// TIA Portal project "Pepsi_Kem_SindelTCU_2024" (V18)
// Pepsi PID ile calisan akis yonlendirme

(* hardware
DEVICE "S7-1200 station_1"  S7-1200 Station
   slot 0: "Rack_0"  S7-1200 Rack  Rack  V1.0
   slot 1: "PLC_1"  CPU 1215C DC/DC/DC  6ES7 215-1AG40-0XB0  V4.5
   slot 2: "DI 8/DQ 8x24VDC_1"  6ES7 223-1BH32-0XB0  V2.0
   slot 3: "AI 4xTC_1"  SM 1231 AI4 x TC  6ES7 231-5QD32-0XB0  V2.0
DEVICE "GSD device_1"  GSD.Device.PN
   slot 0: "Rack"  Rack  V1.0
   slot 0: "SINAMICS-G120X-PN"  SINAMICS G120X(A) PN V1.0  6SL32xx-xYxxx-xxFx  V1.00
      slot 0: "SINAMICS G120X(A) PN V1.0"  SINAMICS G120X(A) PN V1.0
      slot 1: "PN-IO"  PN-IO
         slot 1: "Port 1"  Port 1
         slot 2: "Port 2"  Port 2
      slot 1: "DRIVE_1"  DRIVE
         slot 0: "Module Access Point"  Module Access Point
         slot 1: "without PROFIsafe"  without PROFIsafe
   slot 2: "Standard telegram 1, PZD-2/2"  Standard telegram 1, PZD-2/2
DEVICE "HMI_1"  KTP400 Basic color PN
   slot 0: "HMI_1"  KTP400 Basic color PN  6AV6 647-0AK11-3AX0  12.0.0.0
   slot 1: "HMI_RT_1"  KTP400 Basic color PN  6AV6 647-0AK11-3AX0  12.0.0.0
   slot 5: "HMI_1.IE_CP_1"  PROFINET Interface  12.0.0.0
      slot 1: "PROFINET Interface_1"  PROFINET Interface
         slot 1: "Port_1"  Port
*)

// ===== PLC "PLC_1"  CPU 1215C DC/DC/DC =====
// protected blocks, not shown: "12_TimeToDint"

VAR_GLOBAL   // PLC tag table "Default tag table"
   "Tag_1" AT %MD200 : Time;
   "Tag_2" AT %M200.0 : Bool;
   "Kalip_Modu" AT %M50.0 : Bool;   // Kalip modu
   "Sirkulasyon Modu" AT %M50.1 : Bool;   // Sirkulasyon modu
   "Seq_KalipVanasi_Kapat" AT %M60.0 : Bool;   // Kalip vanasini kapat
   "Seq_Kalip_Vanasi_Ac" AT %M60.1 : Bool;   // Kalip vanasini ac ve kaliba su gonder
   "System_Byte" AT %MB1 : Byte;
   "FirstScan" AT %M1.0 : Bool;
   "DiagStatusUpdate" AT %M1.1 : Bool;
   "AlwaysTRUE" AT %M1.2 : Bool;
   "AlwaysFALSE" AT %M1.3 : Bool;
   "Clock_Byte" AT %MB0 : Byte;
   "Clock_10Hz" AT %M0.0 : Bool;
   "Clock_5Hz" AT %M0.1 : Bool;
   "Clock_2.5Hz" AT %M0.2 : Bool;
   "Clock_2Hz" AT %M0.3 : Bool;
   "Clock_1.25Hz" AT %M0.4 : Bool;
   "Clock_1Hz" AT %M0.5 : Bool;
   "Clock_0.625Hz" AT %M0.6 : Bool;
   "Clock_0.5Hz" AT %M0.7 : Bool;
   "SuAlmaBaslasin" AT %M2.0 : Bool;   // Su al islemi baslasin
   "Seq_TankVanasi_Ac" AT %M2.1 : Bool;   // 0 - Sirkulasyon | 1- Su al
   "MotorDurdu" AT %M2.2 : Bool;
   "yaslandirmaBaslasin" AT %M2.3 : Bool;
   "Yas_Motor1_kontaktor" AT %M2.4 : Bool;
   "Yas_Motor1_Run" AT %M2.5 : Bool;
   "Yas_Motor2_kontaktor" AT %M3.6 : Bool;
   "Yas_Motor2_Run" AT %M2.6 : Bool;
   "Motor1_kontaktor_Secim1" AT %M2.7 : Bool;
   "Motor1_Run_Secim1" AT %M3.0 : Bool;
   "Motor2_kontaktor_Secim2" AT %M3.1 : Bool;
   "Motor2_Run_Secim2" AT %M3.2 : Bool;
   "PID_Setpoint" AT %MD4 : Real;
   "PID_Mode" AT %MW8 : Int;
   "IsiKontroluBaslasin" AT %M3.3 : Bool;
   "TimeET_demo" AT %MD80 : Time;
   "demoStart" AT %M3.4 : Bool;
   "PID_Tunning_Start" AT %M3.5 : Bool;
   "PID_Manuel_Setpoint" AT %MD10 : Real;
   "BOS" AT %M3.7 : Bool;
   "AlarmSusturSet" AT %M14.0 : Bool;
   "tTermikAtti_AlarmSustur" AT %M14.1 : Bool;
   "Man_Tank_SirDolumVan_Ac" AT %M14.2 : Bool;
   "Man_SirKalip_Van_Kapat" AT %M14.3 : Bool;
   "Man_SirKalip_Van_Ac" AT %M14.4 : Bool;
   "Man_Baypass_Van_Kapat" AT %M14.5 : Bool;
   "Man_Baypass_Van_Ac" AT %M14.6 : Bool;
   "Man_Baypass2_Van_Kapat" AT %M14.7 : Bool;
   "Man_Baypass2_Van_Ac" AT %M15.0 : Bool;
   "Man_Motor1_Run" AT %M15.1 : Bool;
   "Man_Motor2_Run" AT %M15.2 : Bool;
   "Man_Motor1_Kontaktor" AT %M15.3 : Bool;
   "Man_Motor2_Kontaktor" AT %M15.4 : Bool;
   "PID_ModeActive_Auto_Edge" AT %M15.5 : Bool;
   "PID_ModeActive_Man_Edge" AT %M15.6 : Bool;
   "BOS_2" AT %M15.7 : Bool;
   "PID_ModeActive_Edge" AT %M16.0 : Bool;
END_VAR

VAR_GLOBAL   // PLC tag table "Drive"
   "axisOFF1_On" AT %M20.0 : Bool;
   "axisAckError" AT %M20.1 : Bool;
   "axisSpeedSp" AT %MD100 : Real;
   "axisRefSpeed" AT %MD104 : Real;
   "axisHWIDSTW" AT %MW50 : Hw_Io;
   "axisHWIDZSW" AT %MW52 : Hw_Io;
   "axisEnabled" AT %M30.0 : Bool;
   "axisLockout" AT %M30.1 : Bool;
   "axisActVelocity" AT %MD120 : Real;
   "axisError" AT %M30.2 : Bool;
   "axisStatus" AT %MW60 : Word;
   "axisDiagId" AT %MW62 : Word;
END_VAR

VAR_GLOBAL CONSTANT   // PLC tag table "LAcycCom_Common"
   "LACYCCOM_BUFFER_ELEMENTS_UPPER_LIM" : Int := 59;   // Upper limit of request buffer array
END_VAR

VAR_GLOBAL CONSTANT   // PLC tag table "LAcycCom_Drives"
   "LACYCCOM_WRITE_PARAMETERS_UPPER_LIM" : Int := 18;   // Upper limit of write parameters
   "LACYCCOM_READ_PARAMETERS_UPPER_LIM" : Int := 38;   // Upper limit of read parameters
   "LACYCCOM_SILENT_OPERATION_PARAMETERS_UPPER_LIM" : Int := 17;   // Upper limit of parameters in LAcycCom_typeDriveSilentOperation
   "LACYCCOM_NO_COMMAND" : Byte := 16#00;   // No command
   "LACYCCOM_READ_COMMAND" : Byte := 16#01;   // Read command
   "LACYCCOM_WRITE_COMMAND" : Byte := 16#02;   // Write command
   "LACYCCOM_TYPE_ALARM" : SInt := 1;   // Alarm
   "LACYCCOM_TYPE_FAULT" : SInt := 2;   // Fault
   "LACYCCOM_TYPE_SI_MESSAGE" : SInt := 3;   // SI message
   "LACYCCOM_MESSAGES_UPPER_LIM" : Int := 23;   // Upper limit of elements in LAcycCom_typeDriveMessages (fix value)
END_VAR

VAR_GLOBAL   // PLC tag table "IO_INPUT"
   "IN_Acil_stop" AT %I0.0 : Bool;
   "IN_Termik" AT %I0.1 : Bool;
   "IN_Tank_Max" AT %I0.2 : Bool;
   "IN_Tank_Min" AT %I0.3 : Bool;
   "IN_Akis_Valfi" AT %IW64 : Int;   // -- AI 0
   "IN_Giris_Sicakligi" AT %IW96 : Int;   // -- TC 0
   "IN_Cikis_Sicakligi" AT %IW98 : Int;   // -- TC 1
   "IN_Tank_SirkulasyonVeDolumVanasi_Kapali" AT %I0.4 : Bool;
   "IN_Tank_SirkulasyonVeDolumVanasi_Acik" AT %I0.5 : Bool;
   "IN_SirkulasyonVeKalipVanasi_Kapali" AT %I0.6 : Bool;
   "IN_SirkulasyonVeKalipVanasi_Acik" AT %I0.7 : Bool;
   "IN_BaypassVanasi_Kapali" AT %I1.0 : Bool;
   "IN_BaypassVanasi_Acik" AT %I1.1 : Bool;
   "IN_UnknownVana_Kapali" AT %I1.2 : Bool;
   "IN_UnknownVana_Acik" AT %I1.3 : Bool;
   "IN_Remote_Calisiyor" AT %I1.4 : Bool;   // karsi taraftan gelen bilgi
   "IN_Remote_Istek" AT %I1.5 : Bool;   // karsi taraftan gelen kaliba gönder bilgisi
END_VAR

VAR_GLOBAL   // PLC tag table "IO_OUTPUT"
   "OUT_Motor1_Kontaktor" AT %Q0.0 : Bool;   // QK1
   "OUT_Motor2_Kontaktor" AT %Q0.1 : Bool;   // QK2
   "OUT_Tank_SirkulasyonVeDolumVanasi" AT %Q0.2 : Bool;   // V101
   "OUT_SirkulasyonVeKalipVanasi_Kapali" AT %Q0.4 : Bool;   // V201
   "OUT_SirkulasyonVeKalipVanasi_Acik" AT %Q0.5 : Bool;   // V202
   "OUT_BaypassVanasi_Kapali" AT %Q0.6 : Bool;   // V301
   "OUT_BaypassVanasi_Acik" AT %Q0.7 : Bool;   // V302
   "OUT_UnknownVana_Kapali" AT %Q1.0 : Bool;   // V401
   "OUT_UnknownVana_Acik" AT %Q1.1 : Bool;   // V402
   "OUT_Lamba_Yesil" AT %Q2.4 : Bool;
   "OUT_Lamba_Sari" AT %Q2.3 : Bool;
   "OUT_Lamba_Kirmizi" AT %Q2.2 : Bool;
   "OUT_Lamba_Siren" AT %Q2.5 : Bool;
   "OUT_Oransal_Vana" AT %QW64 : Int;
END_VAR

DATA_BLOCK "05_Out_DB"   // DB2
{ S7_Optimized_Access := 'TRUE' }
VERSION : 0.1
// stored: InstanceOfName 05_Out
"05_Out"
BEGIN
END_DATA_BLOCK

DATA_BLOCK "01_Ana Merkez_DB"   // DB3
{ S7_Optimized_Access := 'TRUE' }
VERSION : 0.1
// stored: InstanceOfName 01_Ana Merkez
"01_Ana Merkez"
BEGIN
END_DATA_BLOCK

DATA_BLOCK "04_Manuel_DB"   // DB6
{ S7_Optimized_Access := 'TRUE' }
VERSION : 0.1
// stored: InstanceOfName 04_Manuel
"04_Manuel"
BEGIN
END_DATA_BLOCK

DATA_BLOCK "02_Valf Merkezi_DB"   // DB7
{ S7_Optimized_Access := 'TRUE' }
VERSION : 0.1
// stored: InstanceOfName 02_Valf Merkezi
"02_Valf Merkezi"
BEGIN
END_DATA_BLOCK

DATA_BLOCK "03_Yaslandirma_DB"   // DB8
{ S7_Optimized_Access := 'TRUE' }
VERSION : 0.1
// stored: InstanceOfName 03_Yaslandirma
"03_Yaslandirma"
BEGIN
END_DATA_BLOCK

DATA_BLOCK "07_Alarm_DB"   // DB9
{ S7_Optimized_Access := 'TRUE' }
VERSION : 0.1
// stored: InstanceOfName 07_Alarm
"07_Alarm"
BEGIN
END_DATA_BLOCK

DATA_BLOCK "06_Isı Kontrol Sistemi_DB"   // DB10
{ S7_Optimized_Access := 'TRUE' }
VERSION : 0.1
// stored: InstanceOfName 06_Isı Kontrol Sistemi
"06_Isı Kontrol Sistemi"
BEGIN
END_DATA_BLOCK

// folder: Datablcok

DATA_BLOCK "HMI_Data"   // DB1
{ S7_Optimized_Access := 'TRUE' }
VERSION : 0.1
   VAR
      Buttons : Struct
         Otomatik : Bool;   // otomatik mod
         Manuel : Bool;   // manuel mod
         Start : Bool;   // otomatik mod start
         Stop : Bool;   // otomatik mod stop
         driveAckError : Bool;   // surucu hata reset
         AlarmSustur : Bool;
         ManuelButonlar : Struct
            TankSirDolumVanasi_Ac : Bool;
            SirKalipVanasi_Kapat : Bool;
            SirKalipVanasi_Ac : Bool;
            BaypassVanasi1_Kapat : Bool;
            BaypassVanasi1_Ac : Bool;
            BaypassVanasi2_Kapat : Bool;
            BaypassVanasi2_Ac : Bool;
            Motor1_Run : Bool;
            Motor2_Run : Bool;
         END_STRUCT;
      END_STRUCT;
   END_VAR
   VAR RETAIN
      Datas : Struct
         driveSpeed : Real := 50.0;   // motor istenen hiz
         driveReferenceSp : Real := 100.0;   // motor referans hiz
         istenenYaslandirmaSuresi_saat : Int;   // yaslandirma saat suresi
         istenenYaslandirmaSuresi_dk : Int;   // yaslandirma dakika suresi
         motorTercihi : Byte;   // proses icin motor tercihi
         suAlDelayTime : Time;   // su alma icin bekleme suresi
         IstenenSicaklik : Real;   // Istenen sicaklik
      END_STRUCT;
   END_VAR
   VAR
      Infos : Struct
         AnlikGirisSicakligi : Real;   // Okunan giriş sicaklik
         AnlikCikisSicakligi : Real;   // Okunan cikis sicaklik
         SystemDurumu : String[50] := 'Sistem Basladi';   // Sistem durumu bilgilendirme
         driveError : Bool;   // motor hata var mesajı
         driveEnabled : Bool;   // motor aktif edildi
         driveActVelocity : Real;   // motor anlik hiz
         driveLockout : Bool;   // motor duruyor
         yaslandirmaSuresi_saat : DInt;   // yaslandirma süresi gecen saat suresi
         yaslandirmaSuresi_dk : DInt;   // yaslandirma süresi gecen dakika suresi
         yaslandirmaSuresi_sn : DInt;   // yaslandirma süresi gecen saniye suresi
         yaslandirmaStatus : Struct   // aktif yaslandirma
            sag : Bool;
            sol : Bool;
         END_STRUCT;
         FlowMeterOran : Real;   // Flowmeter akis aciklik orani
         OransalVanaOran : Real;   // Oransal vana aciklik orani
      END_STRUCT;
   END_VAR
BEGIN
END_DATA_BLOCK

DATA_BLOCK "System"   // DB4
{ S7_Optimized_Access := 'TRUE' }
VERSION : 0.1
   VAR
      Auto_Man : Bool;   // 0 - manuel | 1- otomatik
      Step_AnaMerkez : Int;   // Ana calisma modu adim bilgisi
      SysBasladi : Bool;
      YaslandirmaSecimi : Byte;   // Yaslandirma secimi
      Step_Yaslandirma : Byte;   // Yaslandirma islem adimi
      Yaslandirma_Suresi : Time;
      Alarm : Word;   // Alarmlar
   END_VAR
BEGIN
END_DATA_BLOCK

// folder: System blocks/Program resources

DATA_BLOCK "Yas_Motor2_Hold_Timer"   // DB5
{ S7_Optimized_Access := 'TRUE' }
AUTHOR : Simatic
FAMILY : IEC
NAME : IEC_TMR
VERSION : 1.0
// stored: InstanceOfName IEC_TIMER
"IEC_TIMER"
BEGIN
END_DATA_BLOCK

// folder: (top level)

ORGANIZATION_BLOCK "Main"   // OB1, LAD, ProgramCycle
TITLE = "Main Program Sweep (Cycle)"
{ S7_Optimized_Access := 'TRUE' }
VERSION : 0.1
   VAR_INPUT
      Initial_Call : Bool;   // Initial call of this OB
      Remanence : Bool;   // =True, if remanent data are available
   END_VAR
BEGIN

REGION Network 1
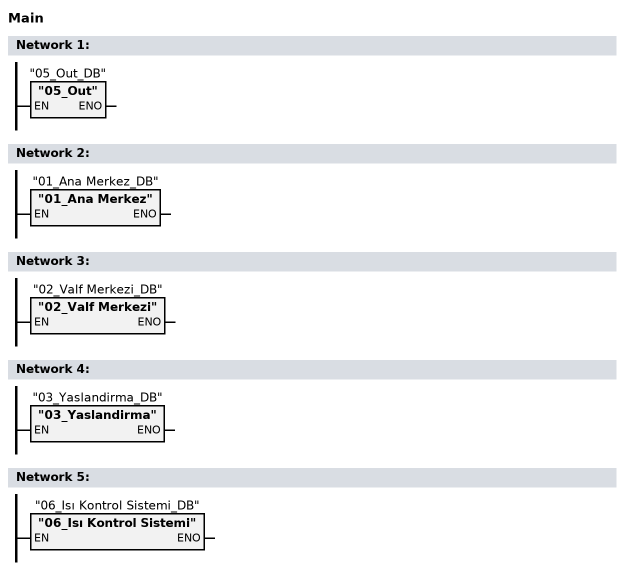
   RUNG wire#powerrail
      "05_Out_DB"()
   END_RUNG
   // the same network as SCL:
   "05_Out_DB"();   // "05_Out"
END_REGION

REGION Network 2
   RUNG wire#powerrail
      "01_Ana Merkez_DB"()
   END_RUNG
   // the same network as SCL:
   "01_Ana Merkez_DB"();   // "01_Ana Merkez"
END_REGION

REGION Network 3
   RUNG wire#powerrail
      "02_Valf Merkezi_DB"()
   END_RUNG
   // the same network as SCL:
   "02_Valf Merkezi_DB"();   // "02_Valf Merkezi"
END_REGION

REGION Network 4
   RUNG wire#powerrail
      "03_Yaslandirma_DB"()
   END_RUNG
   // the same network as SCL:
   "03_Yaslandirma_DB"();   // "03_Yaslandirma"
END_REGION

REGION Network 5
   RUNG wire#powerrail
      "06_Isı Kontrol Sistemi_DB"()
   END_RUNG
   // the same network as SCL:
   "06_Isı Kontrol Sistemi_DB"();   // "06_Isı Kontrol Sistemi"
END_REGION
END_ORGANIZATION_BLOCK

ORGANIZATION_BLOCK "Cyclic interrupt"   // OB30, LAD, CyclicInterrupt
{ S7_Optimized_Access := 'TRUE' }
VERSION : 0.1
   VAR_INPUT
      Initial_Call : Bool;   // Initial call of this OB
      Event_Count : Int;   // Events discarded
   END_VAR
BEGIN

REGION Network 1
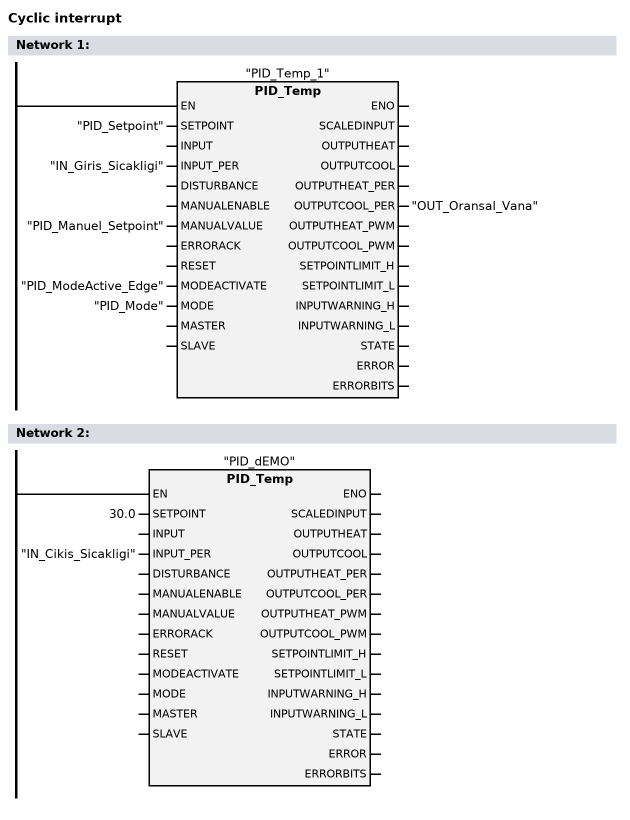
   "PID_Temp_1"(Setpoint := "PID_Setpoint",   // PID_Temp
                Input_PER := "IN_Giris_Sicakligi",
                ManualValue := "PID_Manuel_Setpoint",
                ModeActivate := "PID_ModeActive_Edge",
                Mode := "PID_Mode",
                OutputCool_PER => "OUT_Oransal_Vana");
END_REGION

REGION Network 2
   "PID_dEMO"(Setpoint := 30.0, Input_PER := "IN_Cikis_Sicakligi");   // PID_Temp
END_REGION
END_ORGANIZATION_BLOCK

ORGANIZATION_BLOCK "Diagnostic error interrupt"   // OB82, LAD, DiagnosticErrorInterrupt
{ S7_Optimized_Access := 'TRUE' }
VERSION : 0.1
   VAR_INPUT
      IO_State : Word;   // IO state of the HW object
      LADDR : Hw_Any;   // Hardware identifier
      Channel : UInt;   // Channel number
      MultiError : Bool;   // =true if more than one error is present
   END_VAR
BEGIN
END_ORGANIZATION_BLOCK

ORGANIZATION_BLOCK "Pull or plug of modules"   // OB83, LAD, PullPlug
{ S7_Optimized_Access := 'TRUE' }
VERSION : 0.1
   VAR_INPUT
      LADDR : Hw_Io;   // Hardware identifier
      Event_Class : Byte;   // 16#38/39: module inserted, removed
      Fault_ID : Byte;   // Fault identifier
   END_VAR
BEGIN
END_ORGANIZATION_BLOCK

ORGANIZATION_BLOCK "Rack or station failure"   // OB86, LAD, RackStationFailure
{ S7_Optimized_Access := 'TRUE' }
VERSION : 0.1
   VAR_INPUT
      LADDR : Hw_Device;   // Hardware identifier
      Event_Class : Byte;   // Event class
      Fault_ID : Byte;   // Fault identifier
   END_VAR
BEGIN
END_ORGANIZATION_BLOCK

ORGANIZATION_BLOCK "Task_2"   // OB123, LAD, ProgramCycle
TITLE = "Main Program Sweep (Cycle)"
{ S7_Optimized_Access := 'TRUE' }
VERSION : 0.1
   VAR_INPUT
      Initial_Call : Bool;   // Initial call of this OB
      Remanence : Bool;   // =True, if remanent data are available
   END_VAR
BEGIN

REGION Network 1
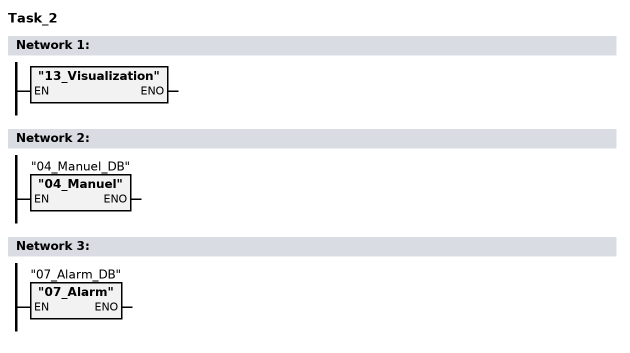
   RUNG wire#powerrail
      "13_Visualization"()
   END_RUNG
   // the same network as SCL:
   "13_Visualization"();
END_REGION

REGION Network 2
   RUNG wire#powerrail
      "04_Manuel_DB"()
   END_RUNG
   // the same network as SCL:
   "04_Manuel_DB"();   // "04_Manuel"
END_REGION

REGION Network 3
   RUNG wire#powerrail
      "07_Alarm_DB"()
   END_RUNG
   // the same network as SCL:
   "07_Alarm_DB"();   // "07_Alarm"
END_REGION
END_ORGANIZATION_BLOCK

// folder: Function

FUNCTION "11_IntToTimer" : Void   // FC1, LAD
{ S7_Optimized_Access := 'TRUE' }
VERSION : 0.1
   VAR_INPUT
      Saat : Int;
      Dakika : Int;
   END_VAR
   VAR_OUTPUT
      HesaplananSure : Time;
   END_VAR
   VAR_TEMP
      tSaat_Dint : DInt;
      tHesaplananSaat : DInt;
      tDakika_Dint : DInt;
      tHesaplananDakika : DInt;
      tHesaplananSure_Dint : DInt;
      tHesaplananSure_Real : Real;
   END_VAR
BEGIN

REGION Network 1
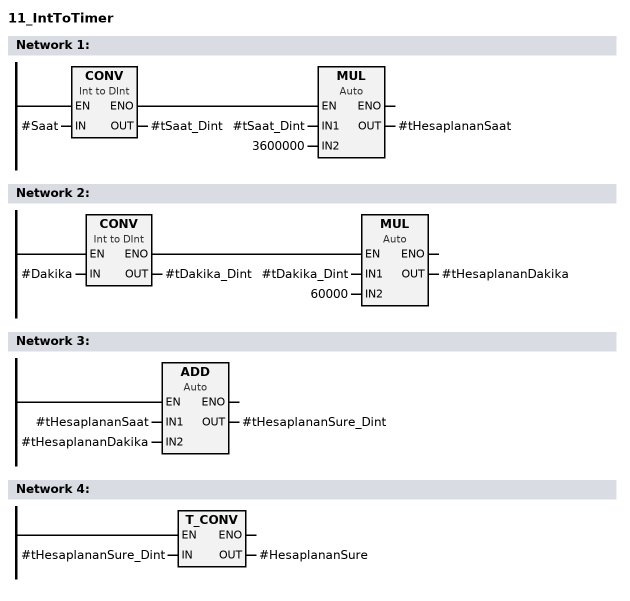
   RUNG wire#powerrail
      { S7_Templates := "[SrcType := Int, DestType := DInt]" } Convert(in := #Saat, out => #tSaat_Dint)
      Mul(in1 := #tSaat_Dint, in2 := 3600000, out => #tHesaplananSaat)
   END_RUNG
   // the same network as SCL:
   #tSaat_Dint := INT_TO_DINT(#Saat);
   #tHesaplananSaat := #tSaat_Dint * 3600000;
END_REGION

REGION Network 2
   RUNG wire#powerrail
      { S7_Templates := "[SrcType := Int, DestType := DInt]" } Convert(in := #Dakika, out => #tDakika_Dint)
      Mul(in1 := #tDakika_Dint, in2 := 60000, out => #tHesaplananDakika)
   END_RUNG
   // the same network as SCL:
   #tDakika_Dint := INT_TO_DINT(#Dakika);
   #tHesaplananDakika := #tDakika_Dint * 60000;
END_REGION

REGION Network 3
   RUNG wire#powerrail
      Add(in1 := #tHesaplananSaat, in2 := #tHesaplananDakika, out => #tHesaplananSure_Dint)
   END_RUNG
   // the same network as SCL:
   #tHesaplananSure_Dint := #tHesaplananSaat + #tHesaplananDakika;
END_REGION

REGION Network 4
   #HesaplananSure := T_CONV(IN := #tHesaplananSure_Dint);
END_REGION
END_FUNCTION

FUNCTION "13_Visualization" : Void   // FC3, LAD
{ S7_Optimized_Access := 'TRUE' }
VERSION : 0.1
// EKRAN BILGILERI VE DONUSUMLERI
   VAR_TEMP
      tGirisSicakligi : Real;
      tCikisSicakligi : Real;
   END_VAR
BEGIN

REGION Network 1 (SCL): Sistem durumu bilgilendirme

   // ana ekran bilgilendirme mesajı
   IF "axisError" THEN
       "HMI_Data".Infos.SystemDurumu := 'Surucu hatasi';
   ELSIF NOT "IN_Termik" THEN
       "HMI_Data".Infos.SystemDurumu := 'Termik hatasi veya 2L+ sigor. kontrol et';
   ELSIF "Kalip_Modu" THEN
       "HMI_Data".Infos.SystemDurumu := 'Kaliba gonderiliyor';
   ELSIF "Sirkulasyon Modu" THEN
       "HMI_Data".Infos.SystemDurumu := 'Sirkulasyon yapiliyor';
   ELSIF NOT "System".Auto_Man THEN
       "HMI_Data".Infos.SystemDurumu := 'Manuel Mod kullanimda';
   END_IF;

   // yaslandirma secimi ekran bilgilendirme
   IF ("System".YaslandirmaSecimi = 0
       AND "System".Step_Yaslandirma = 1)
       OR "System".YaslandirmaSecimi = 1 THEN
       "HMI_Data".Infos.yaslandirmaStatus.sol := true;
       "HMI_Data".Infos.yaslandirmaStatus.sag := FALSE;
   ELSIF ("System".YaslandirmaSecimi = 0
       AND "System".Step_Yaslandirma = 2)
       OR "System".YaslandirmaSecimi = 2 THEN
       "HMI_Data".Infos.yaslandirmaStatus.sol := FALSE;
       "HMI_Data".Infos.yaslandirmaStatus.sag := true;
   END_IF;
END_REGION

REGION Network 2: Akis valfi yuzdesel donusum
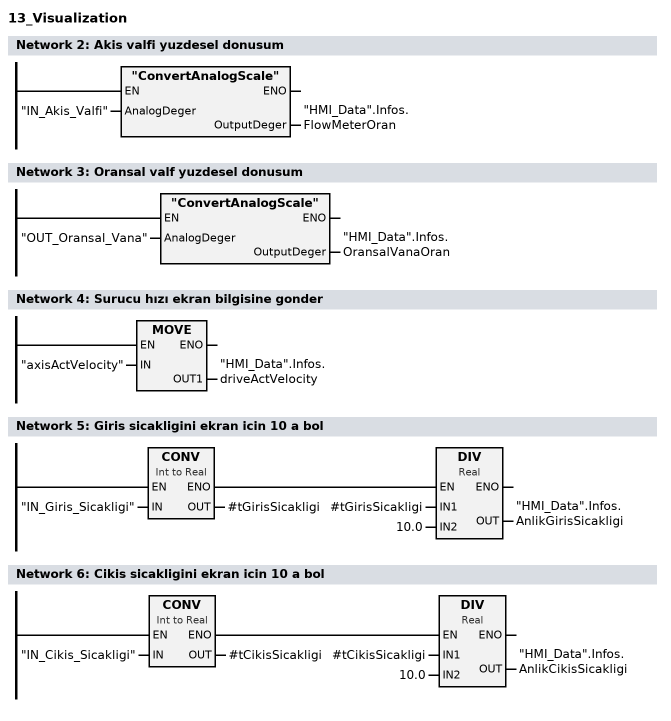
   RUNG wire#powerrail
      "ConvertAnalogScale"(AnalogDeger := "IN_Akis_Valfi", OutputDeger => "HMI_Data".Infos.FlowMeterOran)
   END_RUNG
   // the same network as SCL:
   "ConvertAnalogScale"(AnalogDeger := "IN_Akis_Valfi", OutputDeger => "HMI_Data".Infos.FlowMeterOran);
END_REGION

REGION Network 3: Oransal valf yuzdesel donusum
   RUNG wire#powerrail
      "ConvertAnalogScale"(AnalogDeger := "OUT_Oransal_Vana", OutputDeger => "HMI_Data".Infos.OransalVanaOran)
   END_RUNG
   // the same network as SCL:
   "ConvertAnalogScale"(AnalogDeger := "OUT_Oransal_Vana", OutputDeger => "HMI_Data".Infos.OransalVanaOran);
END_REGION

REGION Network 4: Surucu hızı ekran bilgisine gonder
   RUNG wire#powerrail
      Move(in := "axisActVelocity", out1 => "HMI_Data".Infos.driveActVelocity)
   END_RUNG
   // the same network as SCL:
   "HMI_Data".Infos.driveActVelocity := "axisActVelocity";
END_REGION

REGION Network 5: Giris sicakligini ekran icin 10 a bol
   RUNG wire#powerrail
      { S7_Templates := "[SrcType := Int, DestType := Real]" } Convert(in := "IN_Giris_Sicakligi", out => #tGirisSicakligi)
      { S7_Templates := "SrcType := Real" } Div(in1 := #tGirisSicakligi, in2 := 10.0, out => "HMI_Data".Infos.AnlikGirisSicakligi)
   END_RUNG
   // the same network as SCL:
   #tGirisSicakligi := INT_TO_REAL("IN_Giris_Sicakligi");
   "HMI_Data".Infos.AnlikGirisSicakligi := #tGirisSicakligi / 10.0;
END_REGION

REGION Network 6: Cikis sicakligini ekran icin 10 a bol
   RUNG wire#powerrail
      { S7_Templates := "[SrcType := Int, DestType := Real]" } Convert(in := "IN_Cikis_Sicakligi", out => #tCikisSicakligi)
      { S7_Templates := "SrcType := Real" } Div(in1 := #tCikisSicakligi, in2 := 10.0, out => "HMI_Data".Infos.AnlikCikisSicakligi)
   END_RUNG
   // the same network as SCL:
   #tCikisSicakligi := INT_TO_REAL("IN_Cikis_Sicakligi");
   "HMI_Data".Infos.AnlikCikisSicakligi := #tCikisSicakligi / 10.0;
END_REGION
END_FUNCTION

FUNCTION "ConvertAnalogScale" : Void   // FC4, LAD
{ S7_Optimized_Access := 'TRUE' }
VERSION : 0.1
   VAR_INPUT
      AnalogDeger : Int;
   END_VAR
   VAR_OUTPUT
      OutputDeger : Real;
   END_VAR
   VAR_TEMP
      tRealValue : Real;
      tNorm_Result : Real;
   END_VAR
BEGIN

REGION Network 1
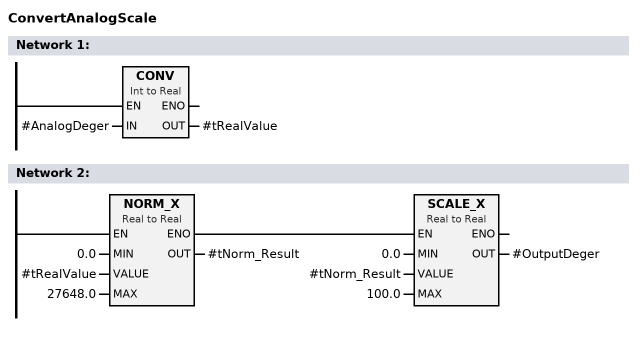
   RUNG wire#powerrail
      { S7_Templates := "[SrcType := Int, DestType := Real]" } Convert(in := #AnalogDeger, out => #tRealValue)
   END_RUNG
   // the same network as SCL:
   #tRealValue := INT_TO_REAL(#AnalogDeger);
END_REGION

REGION Network 2
   RUNG wire#powerrail
      { S7_Templates := "[SrcType := Real, DestType := Real]" } Normalize(min := 0.0, value := #tRealValue, max := 27648.0, out => #tNorm_Result)
      { S7_Templates := "[SrcType := Real, DestType := Real]" } Scale(min := 0.0, value := #tNorm_Result, max := 100.0, out => #OutputDeger)
   END_RUNG
   // the same network as SCL:
   #tNorm_Result := NORM_X(MIN := 0.0, VALUE := #tRealValue, MAX := 27648.0);
   #OutputDeger := SCALE_X(MIN := 0.0, VALUE := #tNorm_Result, MAX := 100.0);
END_REGION
END_FUNCTION

// folder: Function Block

FUNCTION_BLOCK "06_Isı Kontrol Sistemi"   // FB1, LAD
{ S7_Optimized_Access := 'TRUE' }
VERSION : 0.1
// Oransal valfin kontrol edildigi yer
   VAR
      PID_Temp_1 : PID_Temp;
      PID_Compact_1 : PID_Compact;
      ModeActive_M : Bool;
      TP_Timer_Inst : TP_TIME;
      IEC_Timer_0_Instance : TON_TIME;
      IEC_Timer_0_Instance_1 : TP_TIME;
   END_VAR
   VAR_TEMP   // added for the SCL form of the ladder/FBD networks
      _w1 : Bool;
   END_VAR
   // PID_Temp_1.Mode := 4;
BEGIN

REGION Network 1: Oransal valf baslama sarti
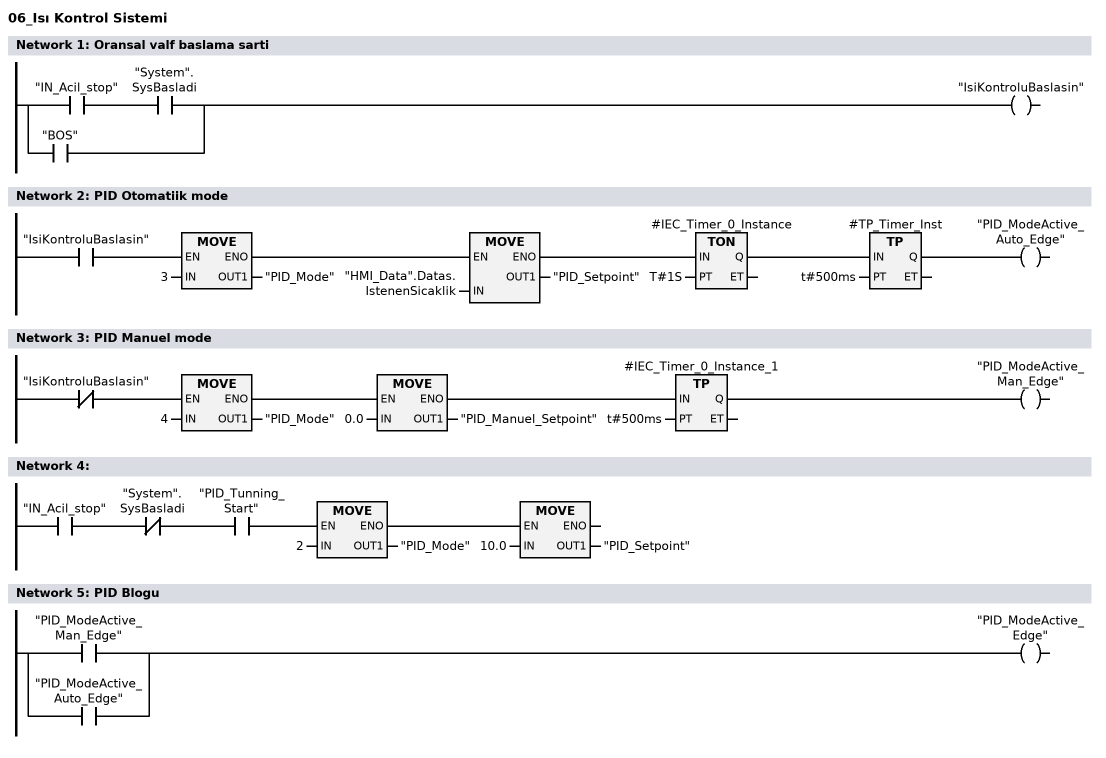
   RUNG wire#powerrail
      Contact( "IN_Acil_stop" )
      Contact( "System".SysBasladi )
      wire#w1
      Coil( "IsiKontroluBaslasin" )
   END_RUNG
   RUNG wire#powerrail
      Contact( "BOS" )
   END_RUNG wire#w1
   // the same network as SCL:
   "IsiKontroluBaslasin" := ("IN_Acil_stop" AND "System".SysBasladi) OR "BOS";
END_REGION

REGION Network 2: PID Otomatiik mode
   IF "IsiKontroluBaslasin" THEN
       "PID_Mode" := 3;
       "PID_Setpoint" := "HMI_Data".Datas.IstenenSicaklik;
   END_IF;
   #IEC_Timer_0_Instance(IN := "IsiKontroluBaslasin", PT := T#1S);   // TON
   #TP_Timer_Inst(IN := #IEC_Timer_0_Instance.Q, PT := t#500ms);   // TP
   "PID_ModeActive_Auto_Edge" := #TP_Timer_Inst.Q;
END_REGION

REGION Network 3: PID Manuel mode
   #_w1 := NOT "IsiKontroluBaslasin";
   IF #_w1 THEN
       "PID_Mode" := 4;
       "PID_Manuel_Setpoint" := 0.0;
   END_IF;
   #IEC_Timer_0_Instance_1(IN := #_w1, PT := t#500ms);   // TP
   "PID_ModeActive_Man_Edge" := #IEC_Timer_0_Instance_1.Q;
END_REGION

REGION Network 4
   RUNG wire#powerrail
      Contact( "IN_Acil_stop" )
      I_Contact( "System".SysBasladi )
      Contact( "PID_Tunning_Start" )
      Move(in := 2, out1 => "PID_Mode")
      Move(in := 10.0, out1 => "PID_Setpoint")
   END_RUNG
   // the same network as SCL:
   IF "IN_Acil_stop" AND NOT "System".SysBasladi AND "PID_Tunning_Start" THEN
       "PID_Mode" := 2;
       "PID_Setpoint" := 10.0;
   END_IF;
END_REGION

REGION Network 5: PID Blogu
   RUNG wire#powerrail
      Contact( "PID_ModeActive_Man_Edge" )
      wire#w1
      Coil( "PID_ModeActive_Edge" )
   END_RUNG
   RUNG wire#powerrail
      Contact( "PID_ModeActive_Auto_Edge" )
   END_RUNG wire#w1
   // the same network as SCL:
   "PID_ModeActive_Edge" := "PID_ModeActive_Man_Edge" OR "PID_ModeActive_Auto_Edge";
END_REGION
END_FUNCTION_BLOCK

FUNCTION_BLOCK "05_Out"   // FB2, LAD
{ S7_Optimized_Access := 'TRUE' }
VERSION : 0.1
   VAR
      SinaSpeed_Instance : SinaSpeed;
   END_VAR
BEGIN

REGION Network 1: Sürücü durdu
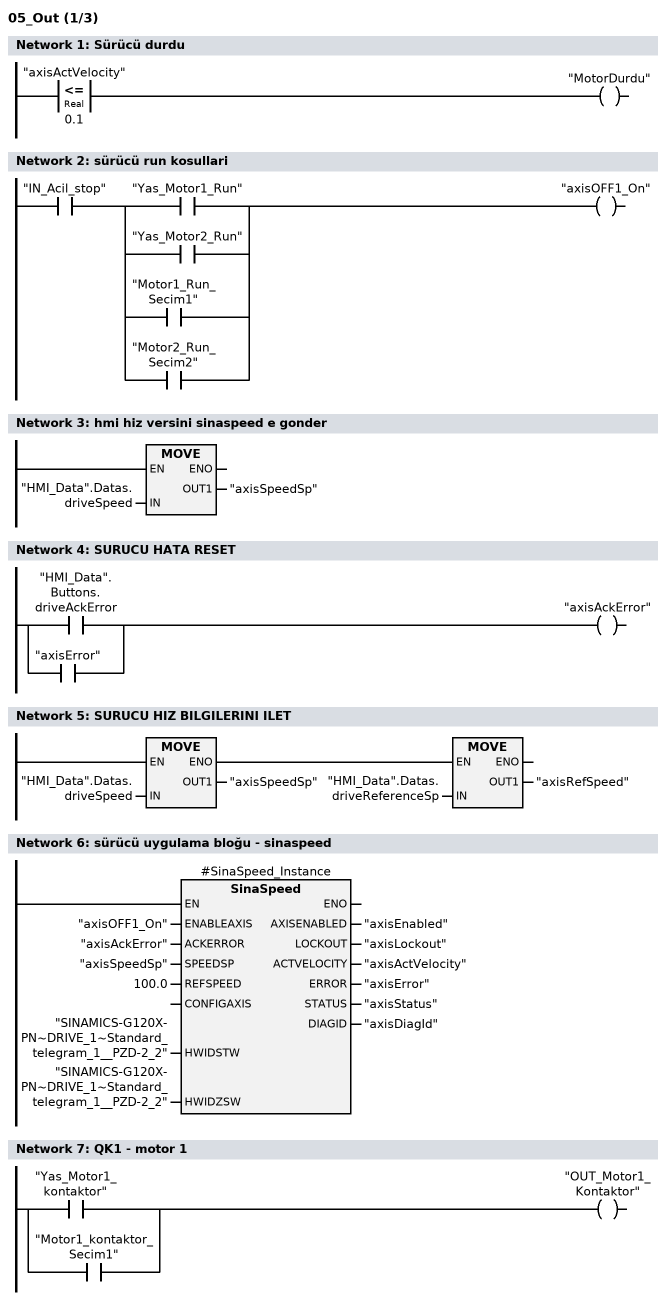
   RUNG wire#powerrail
      { S7_Templates := "SrcType := Real" } LE_Contact(in1 := "axisActVelocity", in2 := 0.1)
      Coil( "MotorDurdu" )
   END_RUNG
   // the same network as SCL:
   "MotorDurdu" := "axisActVelocity" <= 0.1;
END_REGION

REGION Network 2: sürücü run kosullari
   RUNG wire#powerrail
      Contact( "IN_Acil_stop" )
      wire#w1
      Contact( "Yas_Motor1_Run" )
      wire#w2
      Coil( "axisOFF1_On" )
   END_RUNG
   RUNG wire#w1
      Contact( "Yas_Motor2_Run" )
   END_RUNG wire#w2
   RUNG wire#w1
      Contact( "Motor1_Run_Secim1" )
   END_RUNG wire#w2
   RUNG wire#w1
      Contact( "Motor2_Run_Secim2" )
   END_RUNG wire#w2
   // the same network as SCL:
   "axisOFF1_On" := "IN_Acil_stop" AND ("Yas_Motor1_Run" OR "Yas_Motor2_Run" OR "Motor1_Run_Secim1" OR "Motor2_Run_Secim2");
END_REGION

REGION Network 3: hmi hiz versini sinaspeed e gonder
   RUNG wire#powerrail
      Move(in := "HMI_Data".Datas.driveSpeed, out1 => "axisSpeedSp")
   END_RUNG
   // the same network as SCL:
   "axisSpeedSp" := "HMI_Data".Datas.driveSpeed;
END_REGION

REGION Network 4: SURUCU HATA RESET
   RUNG wire#powerrail
      Contact( "HMI_Data".Buttons.driveAckError )
      wire#w1
      Coil( "axisAckError" )
   END_RUNG
   RUNG wire#powerrail
      Contact( "axisError" )
   END_RUNG wire#w1
   // the same network as SCL:
   "axisAckError" := "HMI_Data".Buttons.driveAckError OR "axisError";
END_REGION

REGION Network 5: SURUCU HIZ BILGILERINI ILET
   RUNG wire#powerrail
      Move(in := "HMI_Data".Datas.driveSpeed, out1 => "axisSpeedSp")
      Move(in := "HMI_Data".Datas.driveReferenceSp, out1 => "axisRefSpeed")
   END_RUNG
   // the same network as SCL:
   "axisSpeedSp" := "HMI_Data".Datas.driveSpeed;
   "axisRefSpeed" := "HMI_Data".Datas.driveReferenceSp;
END_REGION

REGION Network 6: sürücü uygulama bloğu - sinaspeed
   #SinaSpeed_Instance(EnableAxis := "axisOFF1_On",   // SinaSpeed
                       AckError := "axisAckError",
                       SpeedSp := "axisSpeedSp",
                       RefSpeed := 100.0,
                       HWIDSTW := "SINAMICS-G120X-PN~DRIVE_1~Standard_telegram_1__PZD-2_2",
                       HWIDZSW := "SINAMICS-G120X-PN~DRIVE_1~Standard_telegram_1__PZD-2_2",
                       AxisEnabled => "axisEnabled",
                       Lockout => "axisLockout",
                       ActVelocity => "axisActVelocity",
                       Error => "axisError",
                       Status => "axisStatus",
                       DiagId => "axisDiagId");
END_REGION

REGION Network 7: QK1 - motor 1
   RUNG wire#powerrail
      Contact( "Yas_Motor1_kontaktor" )
      wire#w1
      Coil( "OUT_Motor1_Kontaktor" )
   END_RUNG
   RUNG wire#powerrail
      Contact( "Motor1_kontaktor_Secim1" )
   END_RUNG wire#w1
   // the same network as SCL:
   "OUT_Motor1_Kontaktor" := "Yas_Motor1_kontaktor" OR "Motor1_kontaktor_Secim1";
END_REGION

REGION Network 8: QK2 - motor 2
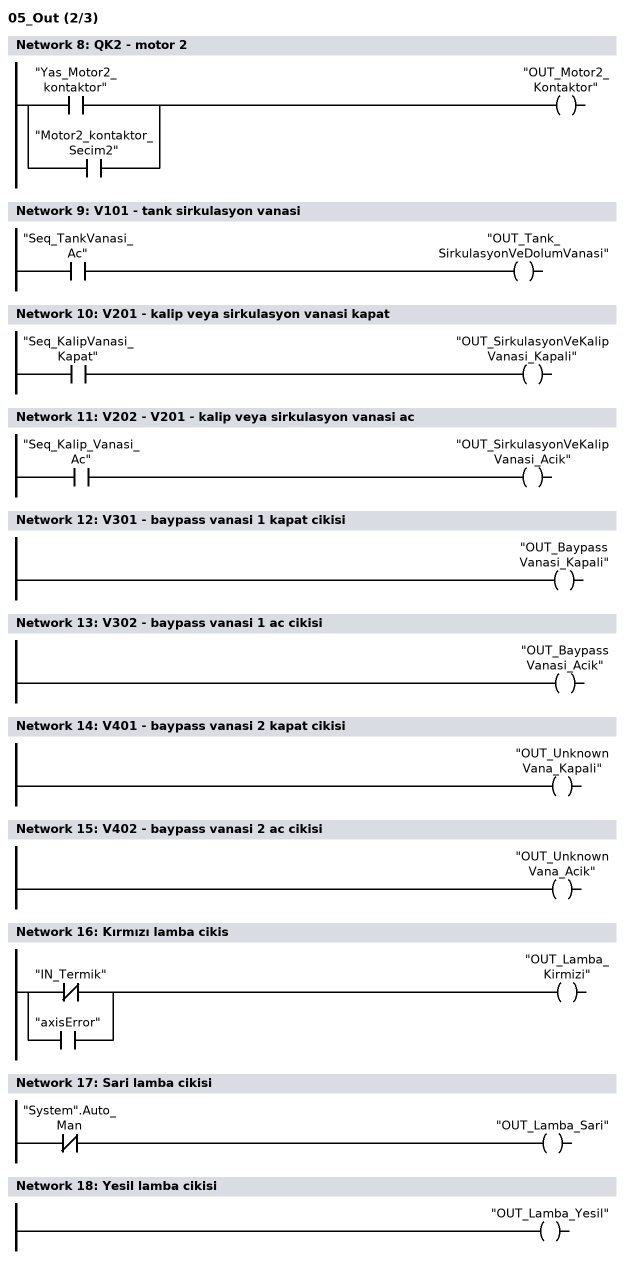
   RUNG wire#powerrail
      Contact( "Yas_Motor2_kontaktor" )
      wire#w1
      Coil( "OUT_Motor2_Kontaktor" )
   END_RUNG
   RUNG wire#powerrail
      Contact( "Motor2_kontaktor_Secim2" )
   END_RUNG wire#w1
   // the same network as SCL:
   "OUT_Motor2_Kontaktor" := "Yas_Motor2_kontaktor" OR "Motor2_kontaktor_Secim2";
END_REGION

REGION Network 9: V101 - tank sirkulasyon vanasi
   RUNG wire#powerrail
      Contact( "Seq_TankVanasi_Ac" )
      Coil( "OUT_Tank_SirkulasyonVeDolumVanasi" )
   END_RUNG
   // the same network as SCL:
   "OUT_Tank_SirkulasyonVeDolumVanasi" := "Seq_TankVanasi_Ac";
END_REGION

REGION Network 10: V201 - kalip veya sirkulasyon vanasi kapat
   RUNG wire#powerrail
      Contact( "Seq_KalipVanasi_Kapat" )
      Coil( "OUT_SirkulasyonVeKalipVanasi_Kapali" )
   END_RUNG
   // the same network as SCL:
   "OUT_SirkulasyonVeKalipVanasi_Kapali" := "Seq_KalipVanasi_Kapat";
END_REGION

REGION Network 11: V202 - V201 - kalip veya sirkulasyon vanasi ac
   RUNG wire#powerrail
      Contact( "Seq_Kalip_Vanasi_Ac" )
      Coil( "OUT_SirkulasyonVeKalipVanasi_Acik" )
   END_RUNG
   // the same network as SCL:
   "OUT_SirkulasyonVeKalipVanasi_Acik" := "Seq_Kalip_Vanasi_Ac";
END_REGION

REGION Network 12: V301 - baypass vanasi 1 kapat cikisi
   RUNG wire#powerrail
      Coil( "OUT_BaypassVanasi_Kapali" )
   END_RUNG
   // the same network as SCL:
   "OUT_BaypassVanasi_Kapali" := TRUE;
END_REGION

REGION Network 13: V302 - baypass vanasi 1 ac cikisi
   RUNG wire#powerrail
      Coil( "OUT_BaypassVanasi_Acik" )
   END_RUNG
   // the same network as SCL:
   "OUT_BaypassVanasi_Acik" := TRUE;
END_REGION

REGION Network 14: V401 - baypass vanasi 2 kapat cikisi
   RUNG wire#powerrail
      Coil( "OUT_UnknownVana_Kapali" )
   END_RUNG
   // the same network as SCL:
   "OUT_UnknownVana_Kapali" := TRUE;
END_REGION

REGION Network 15: V402 - baypass vanasi 2 ac cikisi
   RUNG wire#powerrail
      Coil( "OUT_UnknownVana_Acik" )
   END_RUNG
   // the same network as SCL:
   "OUT_UnknownVana_Acik" := TRUE;
END_REGION

REGION Network 16: Kırmızı lamba cikis
   RUNG wire#powerrail
      I_Contact( "IN_Termik" )
      wire#w1
      Coil( "OUT_Lamba_Kirmizi" )
   END_RUNG
   RUNG wire#powerrail
      Contact( "axisError" )
   END_RUNG wire#w1
   // the same network as SCL:
   "OUT_Lamba_Kirmizi" := NOT "IN_Termik" OR "axisError";
END_REGION

REGION Network 17: Sari lamba cikisi
   RUNG wire#powerrail
      I_Contact( "System".Auto_Man )
      Coil( "OUT_Lamba_Sari" )
   END_RUNG
   // the same network as SCL:
   "OUT_Lamba_Sari" := NOT "System".Auto_Man;
END_REGION

REGION Network 18: Yesil lamba cikisi
   RUNG wire#powerrail
      Coil( "OUT_Lamba_Yesil" )
   END_RUNG
   // the same network as SCL:
   "OUT_Lamba_Yesil" := TRUE;
END_REGION

REGION Network 19: Siren lamba cikisi
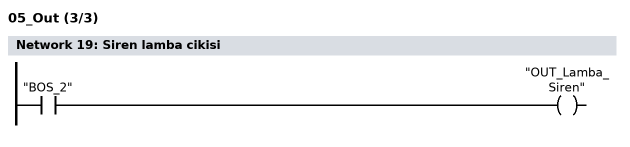
   RUNG wire#powerrail
      Contact( "BOS_2" )
      Coil( "OUT_Lamba_Siren" )
   END_RUNG
   // the same network as SCL:
   "OUT_Lamba_Siren" := "BOS_2";
END_REGION
END_FUNCTION_BLOCK

FUNCTION_BLOCK "07_Alarm"   // FB3, LAD
{ S7_Optimized_Access := 'TRUE' }
VERSION : 0.1
   VAR
      TankDolumVanasi_Inst : TON_TIME;
      KalipDolumVanasi_Inst : TON_TIME;
      BypassVanasi_Inst : TON_TIME;
      BypassVanasi2_Inst : TON_TIME;
      ResetTrig : Bool;
      ResetTrig2 : Bool;
      Manuel_M : Bool;
      Oto_M : Bool;
      Start_M : Bool;
      Stop_M : Bool;
   END_VAR
   VAR_TEMP   // added for the SCL form of the ladder/FBD networks
      _w1 : Bool;
      _w2 : Bool;
      _w3 : Bool;
      _w4 : Bool;
   END_VAR
BEGIN

REGION Network 1: Surucu hata
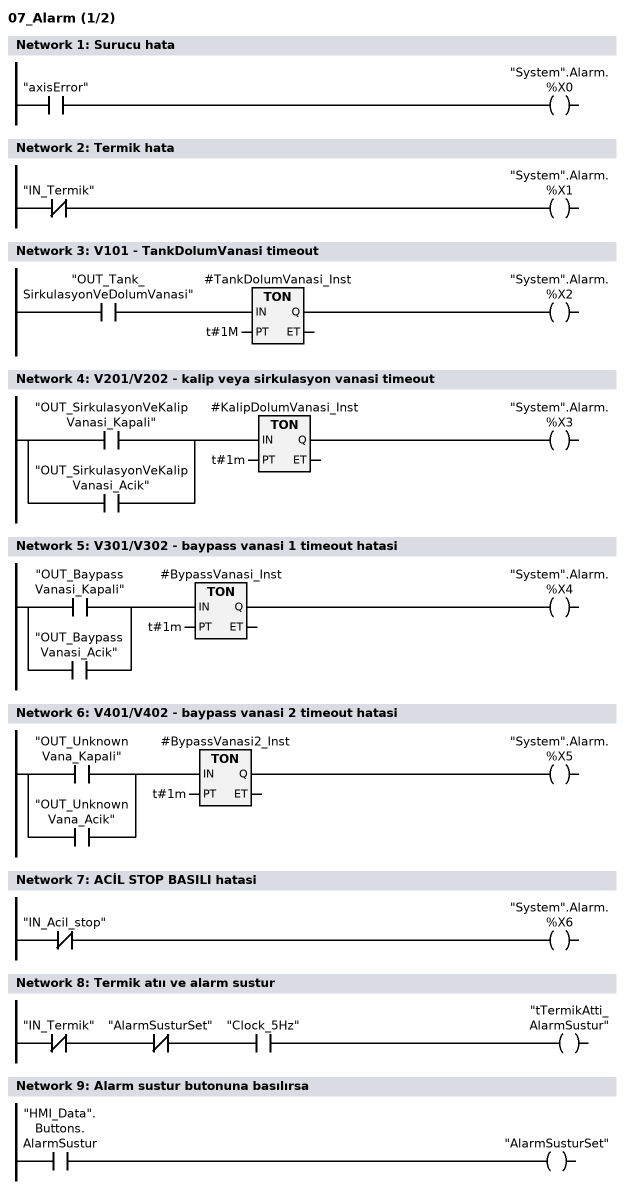
   RUNG wire#powerrail
      Contact( "axisError" )
      Coil( "System".Alarm.%X0 )
   END_RUNG
   // the same network as SCL:
   "System".Alarm.%X0 := "axisError";
END_REGION

REGION Network 2: Termik hata
   RUNG wire#powerrail
      I_Contact( "IN_Termik" )
      Coil( "System".Alarm.%X1 )
   END_RUNG
   // the same network as SCL:
   "System".Alarm.%X1 := NOT "IN_Termik";
END_REGION

REGION Network 3: V101 - TankDolumVanasi timeout
   #TankDolumVanasi_Inst(IN := "OUT_Tank_SirkulasyonVeDolumVanasi", PT := t#1M);   // TON
   "System".Alarm.%X2 := #TankDolumVanasi_Inst.Q;
END_REGION

REGION Network 4: V201/V202 - kalip veya sirkulasyon vanasi timeout
   #KalipDolumVanasi_Inst(IN := "OUT_SirkulasyonVeKalipVanasi_Kapali" OR "OUT_SirkulasyonVeKalipVanasi_Acik",   // TON
                          PT := t#1m);
   "System".Alarm.%X3 := #KalipDolumVanasi_Inst.Q;
END_REGION

REGION Network 5: V301/V302 - baypass vanasi 1 timeout hatasi
   #BypassVanasi_Inst(IN := "OUT_BaypassVanasi_Kapali" OR "OUT_BaypassVanasi_Acik", PT := t#1m);   // TON
   "System".Alarm.%X4 := #BypassVanasi_Inst.Q;
END_REGION

REGION Network 6: V401/V402 - baypass vanasi 2 timeout hatasi
   #BypassVanasi2_Inst(IN := "OUT_UnknownVana_Kapali" OR "OUT_UnknownVana_Acik", PT := t#1m);   // TON
   "System".Alarm.%X5 := #BypassVanasi2_Inst.Q;
END_REGION

REGION Network 7: ACİL STOP BASILI hatasi
   RUNG wire#powerrail
      I_Contact( "IN_Acil_stop" )
      Coil( "System".Alarm.%X6 )
   END_RUNG
   // the same network as SCL:
   "System".Alarm.%X6 := NOT "IN_Acil_stop";
END_REGION

REGION Network 8: Termik atıı ve alarm sustur
   RUNG wire#powerrail
      I_Contact( "IN_Termik" )
      I_Contact( "AlarmSusturSet" )
      Contact( "Clock_5Hz" )
      Coil( "tTermikAtti_AlarmSustur" )
   END_RUNG
   // the same network as SCL:
   "tTermikAtti_AlarmSustur" := NOT "IN_Termik" AND NOT "AlarmSusturSet" AND "Clock_5Hz";
END_REGION

REGION Network 9: Alarm sustur butonuna basılırsa
   RUNG wire#powerrail
      Contact( "HMI_Data".Buttons.AlarmSustur )
      Coil( "AlarmSusturSet" )
   END_RUNG
   // the same network as SCL:
   "AlarmSusturSet" := "HMI_Data".Buttons.AlarmSustur;
END_REGION

REGION Network 10: Alarm sustur bitini resetle
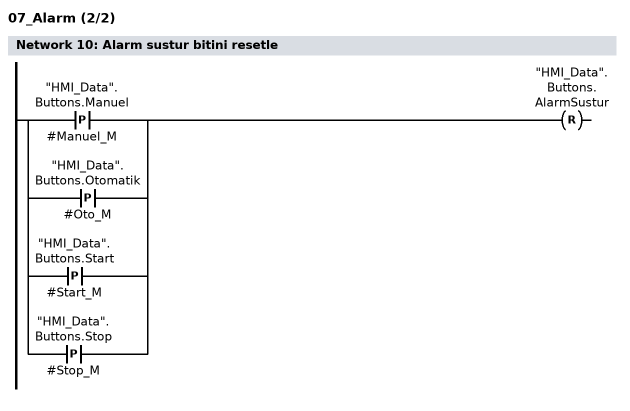
   RUNG wire#powerrail
      P_Contact(operand := "HMI_Data".Buttons.Manuel, bit := #Manuel_M)
      wire#w1
      R_Coil( "HMI_Data".Buttons.AlarmSustur )
   END_RUNG
   RUNG wire#powerrail
      P_Contact(operand := "HMI_Data".Buttons.Otomatik, bit := #Oto_M)
   END_RUNG wire#w1
   RUNG wire#powerrail
      P_Contact(operand := "HMI_Data".Buttons.Start, bit := #Start_M)
   END_RUNG wire#w1
   RUNG wire#powerrail
      P_Contact(operand := "HMI_Data".Buttons.Stop, bit := #Stop_M)
   END_RUNG wire#w1
   // the same network as SCL:
   #_w1 := "HMI_Data".Buttons.Manuel AND NOT #Manuel_M;   // rising edge of "HMI_Data".Buttons.Manuel
   #Manuel_M := "HMI_Data".Buttons.Manuel;
   #_w2 := "HMI_Data".Buttons.Otomatik AND NOT #Oto_M;   // rising edge of "HMI_Data".Buttons.Otomatik
   #Oto_M := "HMI_Data".Buttons.Otomatik;
   #_w3 := "HMI_Data".Buttons.Start AND NOT #Start_M;   // rising edge of "HMI_Data".Buttons.Start
   #Start_M := "HMI_Data".Buttons.Start;
   #_w4 := "HMI_Data".Buttons.Stop AND NOT #Stop_M;   // rising edge of "HMI_Data".Buttons.Stop
   #Stop_M := "HMI_Data".Buttons.Stop;
   IF #_w1 OR #_w2 OR #_w3 OR #_w4 THEN "HMI_Data".Buttons.AlarmSustur := FALSE; END_IF;
END_REGION
END_FUNCTION_BLOCK

FUNCTION_BLOCK "01_Ana Merkez"   // FB4, LAD
{ S7_Optimized_Access := 'TRUE' }
VERSION : 0.1
BEGIN

REGION Network 1
   // otomatik baslama icin gerekli kontroller
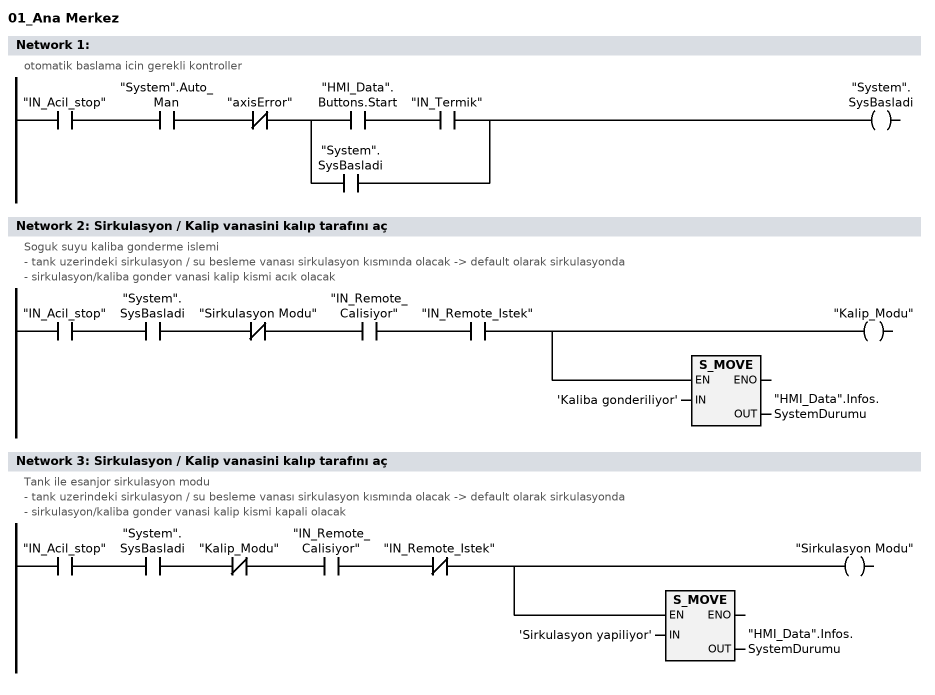
   RUNG wire#powerrail
      Contact( "IN_Acil_stop" )
      Contact( "System".Auto_Man )
      I_Contact( "axisError" )
      wire#w1
      Contact( "HMI_Data".Buttons.Start )
      Contact( "IN_Termik" )
      wire#w2
      Coil( "System".SysBasladi )
   END_RUNG
   RUNG wire#w1
      Contact( "System".SysBasladi )
   END_RUNG wire#w2
   // the same network as SCL:
   "System".SysBasladi := "IN_Acil_stop" AND "System".Auto_Man AND NOT "axisError" AND (("HMI_Data".Buttons.Start AND "IN_Termik") OR "System".SysBasladi);
END_REGION

REGION Network 2: Sirkulasyon / Kalip vanasini kalıp tarafını aç
   // Soguk suyu kaliba gonderme islemi
   // - tank uzerindeki sirkulasyon / su besleme vanası sirkulasyon kısmında olacak -> default olarak sirkulasyonda
   // - sirkulasyon/kaliba gonder vanasi kalip kismi acık olacak
   RUNG wire#powerrail
      Contact( "IN_Acil_stop" )
      Contact( "System".SysBasladi )
      I_Contact( "Sirkulasyon Modu" )
      Contact( "IN_Remote_Calisiyor" )
      Contact( "IN_Remote_Istek" )
      wire#w1
      Coil( "Kalip_Modu" )
   END_RUNG
   RUNG wire#w1
      S_Move(in := 'Kaliba gonderiliyor', out => "HMI_Data".Infos.SystemDurumu)
   END_RUNG
   // the same network as SCL:
   "Kalip_Modu" := "IN_Acil_stop" AND "System".SysBasladi AND NOT "Sirkulasyon Modu" AND "IN_Remote_Calisiyor" AND "IN_Remote_Istek";
   IF "Kalip_Modu" THEN "HMI_Data".Infos.SystemDurumu := 'Kaliba gonderiliyor'; END_IF;
END_REGION

REGION Network 3: Sirkulasyon / Kalip vanasini kalıp tarafını aç
   // Tank ile esanjor sirkulasyon modu
   // - tank uzerindeki sirkulasyon / su besleme vanası sirkulasyon kısmında olacak -> default olarak sirkulasyonda
   // - sirkulasyon/kaliba gonder vanasi kalip kismi kapali olacak
   RUNG wire#powerrail
      Contact( "IN_Acil_stop" )
      Contact( "System".SysBasladi )
      I_Contact( "Kalip_Modu" )
      Contact( "IN_Remote_Calisiyor" )
      I_Contact( "IN_Remote_Istek" )
      wire#w1
      Coil( "Sirkulasyon Modu" )
   END_RUNG
   RUNG wire#w1
      S_Move(in := 'Sirkulasyon yapiliyor', out => "HMI_Data".Infos.SystemDurumu)
   END_RUNG
   // the same network as SCL:
   "Sirkulasyon Modu" := "IN_Acil_stop" AND "System".SysBasladi AND NOT "Kalip_Modu" AND "IN_Remote_Calisiyor" AND NOT "IN_Remote_Istek";
   IF "Sirkulasyon Modu" THEN "HMI_Data".Infos.SystemDurumu := 'Sirkulasyon yapiliyor'; END_IF;
END_REGION
END_FUNCTION_BLOCK

FUNCTION_BLOCK "02_Valf Merkezi"   // FB5, LAD
{ S7_Optimized_Access := 'TRUE' }
VERSION : 0.1
// Sirkulasyon Modu vana kontrolleri
// 
// --------------BYPASS VANALARI EKLENECEK---------------------------
   VAR
      SuAlTimer_Inst : TON_TIME;
      SuAlTimer2_Inst : TON_TIME;
   END_VAR
   VAR_TEMP   // added for the SCL form of the ladder/FBD networks
      _w1 : Bool;
   END_VAR
BEGIN

REGION Network 1: Sirkulasyon Modu -> kalip vanasini kapat
   // Kalip vanasi kapali -> sirkulasyon yapar
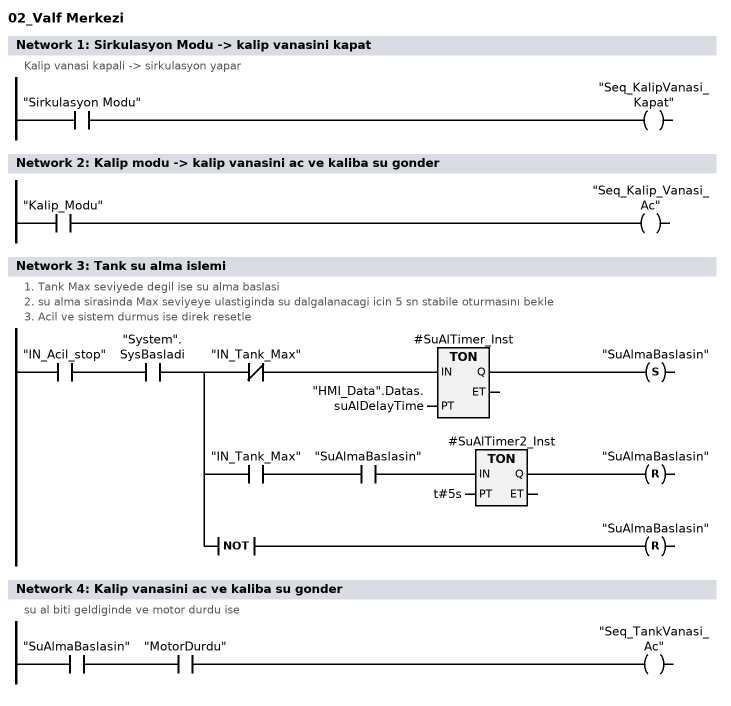
   RUNG wire#powerrail
      Contact( "Sirkulasyon Modu" )
      Coil( "Seq_KalipVanasi_Kapat" )
   END_RUNG
   // the same network as SCL:
   "Seq_KalipVanasi_Kapat" := "Sirkulasyon Modu";
END_REGION

REGION Network 2: Kalip modu -> kalip vanasini ac ve kaliba su gonder
   RUNG wire#powerrail
      Contact( "Kalip_Modu" )
      Coil( "Seq_Kalip_Vanasi_Ac" )
   END_RUNG
   // the same network as SCL:
   "Seq_Kalip_Vanasi_Ac" := "Kalip_Modu";
END_REGION

REGION Network 3: Tank su alma islemi
   // 1. Tank Max seviyede degil ise su alma baslasi
   // 2. su alma sirasinda Max seviyeye ulastiginda su dalgalanacagi icin 5 sn stabile oturmasını bekle
   // 3. Acil ve sistem durmus ise direk resetle
   #_w1 := "IN_Acil_stop" AND "System".SysBasladi;
   #SuAlTimer_Inst(IN := #_w1 AND NOT "IN_Tank_Max", PT := "HMI_Data".Datas.suAlDelayTime);   // TON
   IF #SuAlTimer_Inst.Q THEN "SuAlmaBaslasin" := TRUE; END_IF;
   #SuAlTimer2_Inst(IN := #_w1 AND "IN_Tank_Max" AND "SuAlmaBaslasin", PT := t#5s);   // TON
   IF #SuAlTimer2_Inst.Q THEN "SuAlmaBaslasin" := FALSE; END_IF;
   IF NOT #_w1 THEN "SuAlmaBaslasin" := FALSE; END_IF;
END_REGION

REGION Network 4: Kalip vanasini ac ve kaliba su gonder
   // su al biti geldiginde ve motor durdu ise
   RUNG wire#powerrail
      Contact( "SuAlmaBaslasin" )
      Contact( "MotorDurdu" )
      Coil( "Seq_TankVanasi_Ac" )
   END_RUNG
   // the same network as SCL:
   "Seq_TankVanasi_Ac" := "SuAlmaBaslasin" AND "MotorDurdu";
END_REGION
END_FUNCTION_BLOCK

FUNCTION_BLOCK "03_Yaslandirma"   // FB6, LAD
{ S7_Optimized_Access := 'TRUE' }
VERSION : 0.1
   VAR
      Yas_Motor1_Timer : TON_TIME;
      Yas_Moto1_Hold_Timer : TON_TIME;
      Motor1_Run_Delay : TON_TIME;
      Motor2_Run_Delay : TON_TIME;
      Yas_Motor2_Timer : TON_TIME;
      Yas_Secim1_Motor_Timer : TON_TIME;
      Yas_Secim2_Motor_Timer : TON_TIME;
      IEC_Timer_0_Instance : TON_TIME;
      IEC_Timer_0_Instance_1 : TON_TIME;
   END_VAR
   VAR_TEMP
      Yas_Motor1_TimeET : Time;
      Yas_Motor2_TimeET : Time;
   END_VAR
BEGIN

REGION Network 1: eKRAN SAAT ve DAKIKA degerini TIME 'A DONUSTUR
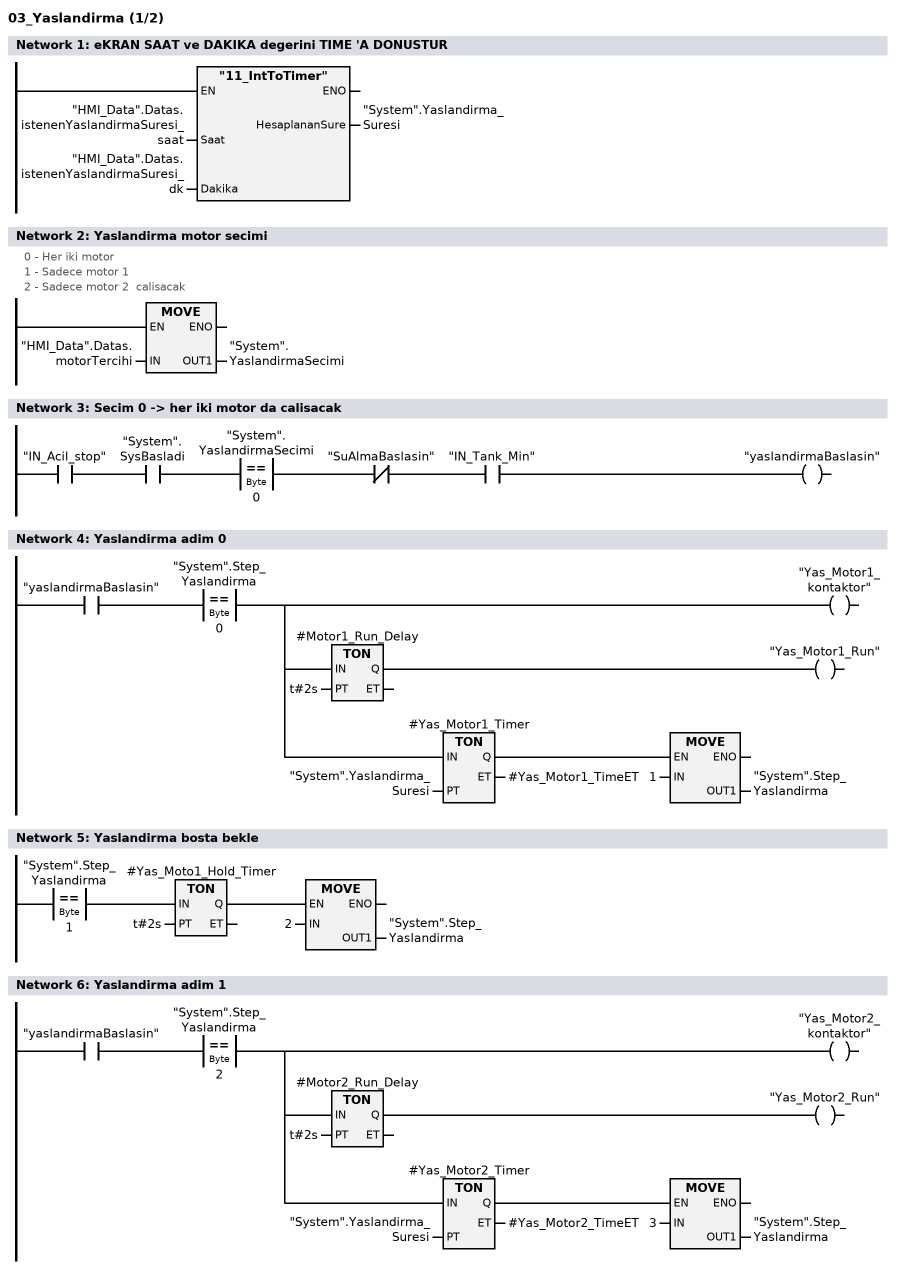
   RUNG wire#powerrail
      "11_IntToTimer"(Saat := "HMI_Data".Datas.istenenYaslandirmaSuresi_saat, Dakika := "HMI_Data".Datas.istenenYaslandirmaSuresi_dk, HesaplananSure => "System".Yaslandirma_Suresi)
   END_RUNG
   // the same network as SCL:
   "11_IntToTimer"(Saat := "HMI_Data".Datas.istenenYaslandirmaSuresi_saat,
                   Dakika := "HMI_Data".Datas.istenenYaslandirmaSuresi_dk,
                   HesaplananSure => "System".Yaslandirma_Suresi);
END_REGION

REGION Network 2: Yaslandirma motor secimi
   // 0 - Her iki motor
   // 1 - Sadece motor 1 
   // 2 - Sadece motor 2  calisacak
   RUNG wire#powerrail
      Move(in := "HMI_Data".Datas.motorTercihi, out1 => "System".YaslandirmaSecimi)
   END_RUNG
   // the same network as SCL:
   "System".YaslandirmaSecimi := "HMI_Data".Datas.motorTercihi;
END_REGION

REGION Network 3: Secim 0 -> her iki motor da calisacak
   RUNG wire#powerrail
      Contact( "IN_Acil_stop" )
      Contact( "System".SysBasladi )
      { S7_Templates := "SrcType := Byte" } EQ_Contact(in1 := "System".YaslandirmaSecimi, in2 := 0)
      I_Contact( "SuAlmaBaslasin" )
      Contact( "IN_Tank_Min" )
      Coil( "yaslandirmaBaslasin" )
   END_RUNG
   // the same network as SCL:
   "yaslandirmaBaslasin" := "IN_Acil_stop" AND "System".SysBasladi AND ("System".YaslandirmaSecimi = 0) AND NOT "SuAlmaBaslasin" AND "IN_Tank_Min";
END_REGION

REGION Network 4: Yaslandirma adim 0
   "Yas_Motor1_kontaktor" := "yaslandirmaBaslasin" AND ("System".Step_Yaslandirma = 0);
   #Motor1_Run_Delay(IN := "Yas_Motor1_kontaktor", PT := t#2s);   // TON
   "Yas_Motor1_Run" := #Motor1_Run_Delay.Q;
   #Yas_Motor1_Timer(IN := "Yas_Motor1_kontaktor", PT := "System".Yaslandirma_Suresi, ET => #Yas_Motor1_TimeET);   // TON
   IF #Yas_Motor1_Timer.Q THEN "System".Step_Yaslandirma := 1; END_IF;
END_REGION

REGION Network 5: Yaslandirma bosta bekle
   #Yas_Moto1_Hold_Timer(IN := "System".Step_Yaslandirma = 1, PT := t#2s);   // TON
   IF #Yas_Moto1_Hold_Timer.Q THEN "System".Step_Yaslandirma := 2; END_IF;
END_REGION

REGION Network 6: Yaslandirma adim 1
   "Yas_Motor2_kontaktor" := "yaslandirmaBaslasin" AND ("System".Step_Yaslandirma = 2);
   #Motor2_Run_Delay(IN := "Yas_Motor2_kontaktor", PT := t#2s);   // TON
   "Yas_Motor2_Run" := #Motor2_Run_Delay.Q;
   #Yas_Motor2_Timer(IN := "Yas_Motor2_kontaktor", PT := "System".Yaslandirma_Suresi, ET => #Yas_Motor2_TimeET);   // TON
   IF #Yas_Motor2_Timer.Q THEN "System".Step_Yaslandirma := 3; END_IF;
END_REGION

REGION Network 7: Yaslandirma bosta bekle
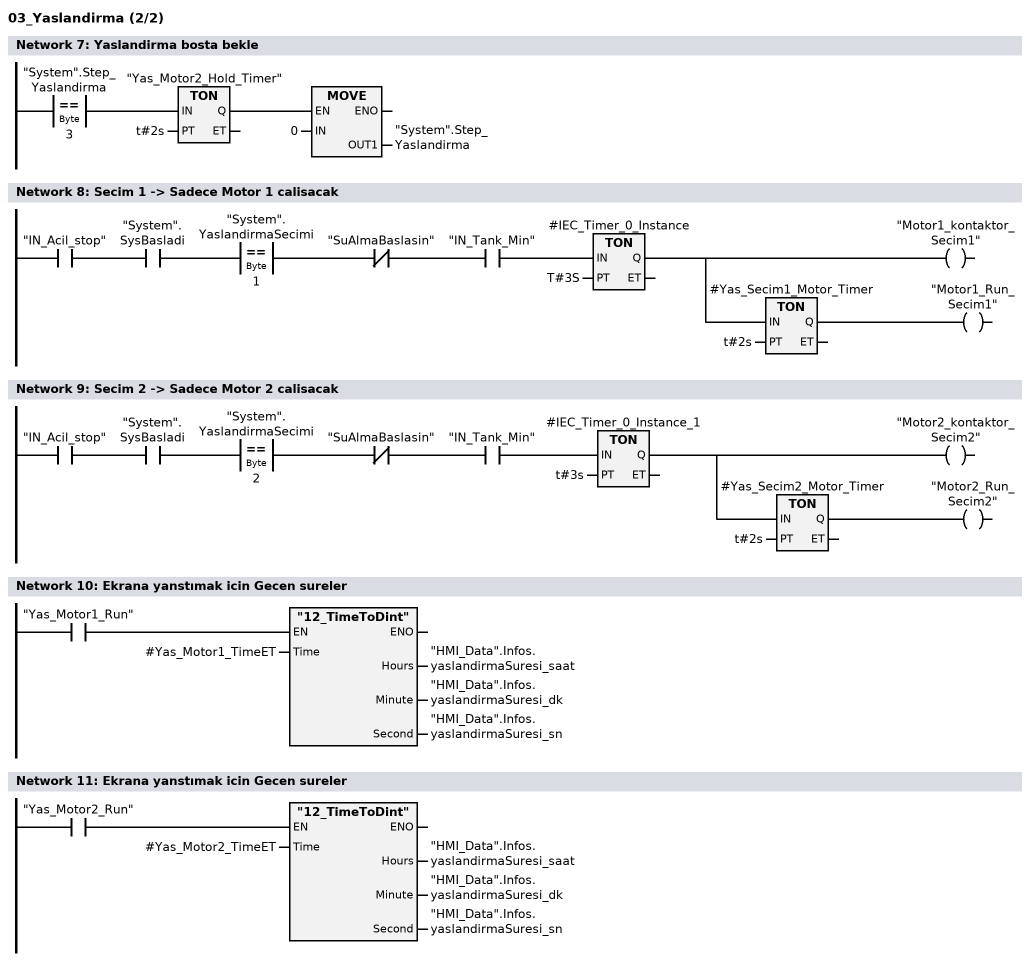
   "Yas_Motor2_Hold_Timer".TON(IN := "System".Step_Yaslandirma = 3, PT := t#2s);
   IF "Yas_Motor2_Hold_Timer".Q THEN "System".Step_Yaslandirma := 0; END_IF;
END_REGION

REGION Network 8: Secim 1 -> Sadece Motor 1 calisacak
   #IEC_Timer_0_Instance(IN := "IN_Acil_stop" AND "System".SysBasladi AND ("System".YaslandirmaSecimi = 1) AND NOT "SuAlmaBaslasin" AND "IN_Tank_Min",   // TON
                         PT := T#3S);
   "Motor1_kontaktor_Secim1" := #IEC_Timer_0_Instance.Q;
   #Yas_Secim1_Motor_Timer(IN := #IEC_Timer_0_Instance.Q, PT := t#2s);   // TON
   "Motor1_Run_Secim1" := #Yas_Secim1_Motor_Timer.Q;
END_REGION

REGION Network 9: Secim 2 -> Sadece Motor 2 calisacak
   #IEC_Timer_0_Instance_1(IN := "IN_Acil_stop" AND "System".SysBasladi AND ("System".YaslandirmaSecimi = 2) AND NOT "SuAlmaBaslasin" AND "IN_Tank_Min",   // TON
                           PT := t#3s);
   "Motor2_kontaktor_Secim2" := #IEC_Timer_0_Instance_1.Q;
   #Yas_Secim2_Motor_Timer(IN := #IEC_Timer_0_Instance_1.Q, PT := t#2s);   // TON
   "Motor2_Run_Secim2" := #Yas_Secim2_Motor_Timer.Q;
END_REGION

REGION Network 10: Ekrana yanstımak icin Gecen sureler
   RUNG wire#powerrail
      Contact( "Yas_Motor1_Run" )
      "12_TimeToDint"("Time" := #Yas_Motor1_TimeET, Hours => "HMI_Data".Infos.yaslandirmaSuresi_saat, Minute => "HMI_Data".Infos.yaslandirmaSuresi_dk, Second => "HMI_Data".Infos.yaslandirmaSuresi_sn)
   END_RUNG
   // the same network as SCL:
   IF "Yas_Motor1_Run" THEN
       "12_TimeToDint"("Time" := #Yas_Motor1_TimeET,
                       Hours => "HMI_Data".Infos.yaslandirmaSuresi_saat,
                       Minute => "HMI_Data".Infos.yaslandirmaSuresi_dk,
                       Second => "HMI_Data".Infos.yaslandirmaSuresi_sn);
   END_IF;
END_REGION

REGION Network 11: Ekrana yanstımak icin Gecen sureler
   RUNG wire#powerrail
      Contact( "Yas_Motor2_Run" )
      "12_TimeToDint"("Time" := #Yas_Motor2_TimeET, Hours => "HMI_Data".Infos.yaslandirmaSuresi_saat, Minute => "HMI_Data".Infos.yaslandirmaSuresi_dk, Second => "HMI_Data".Infos.yaslandirmaSuresi_sn)
   END_RUNG
   // the same network as SCL:
   IF "Yas_Motor2_Run" THEN
       "12_TimeToDint"("Time" := #Yas_Motor2_TimeET,
                       Hours => "HMI_Data".Infos.yaslandirmaSuresi_saat,
                       Minute => "HMI_Data".Infos.yaslandirmaSuresi_dk,
                       Second => "HMI_Data".Infos.yaslandirmaSuresi_sn);
   END_IF;
END_REGION
END_FUNCTION_BLOCK

FUNCTION_BLOCK "04_Manuel"   // FB7, LAD
{ S7_Optimized_Access := 'TRUE' }
VERSION : 0.1
   VAR
      Man_Motor1_Run_Timer : TON_TIME;
      Man_Motor2_Run_Timer : TON_TIME;
   END_VAR
BEGIN

REGION Network 1: Tank sirk. dolum vanasi ac
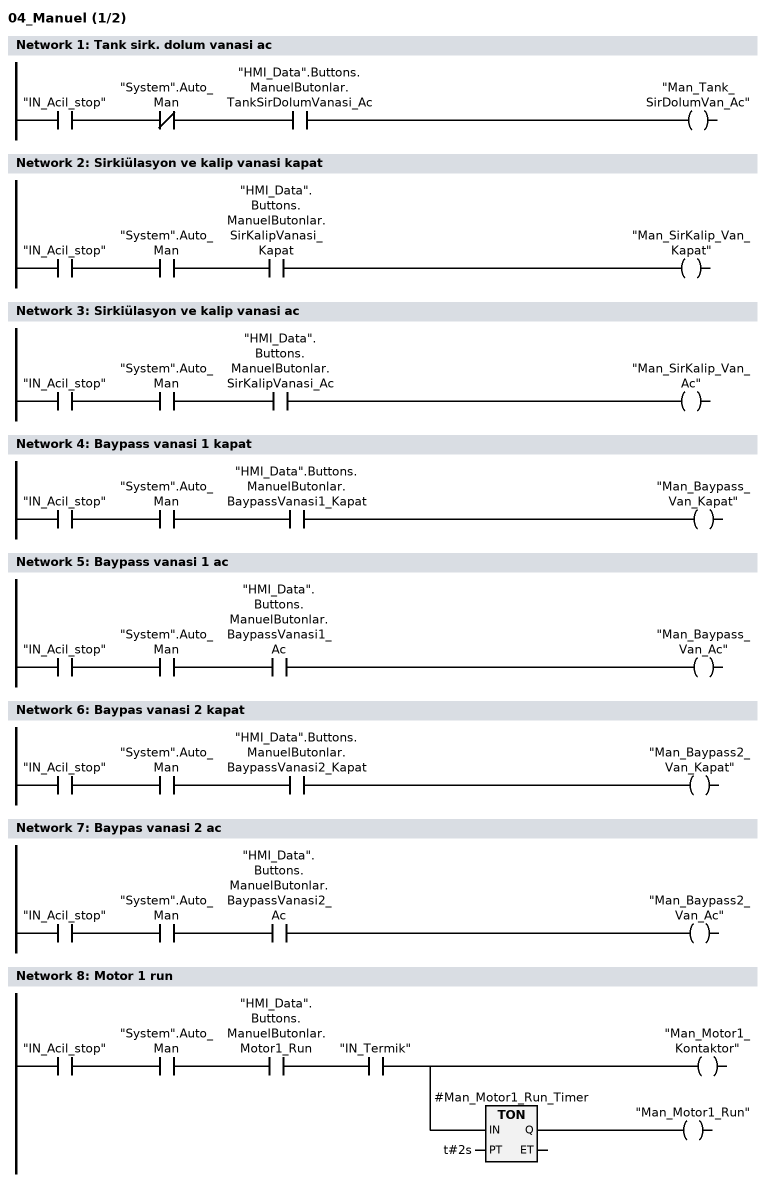
   RUNG wire#powerrail
      Contact( "IN_Acil_stop" )
      I_Contact( "System".Auto_Man )
      Contact( "HMI_Data".Buttons.ManuelButonlar.TankSirDolumVanasi_Ac )
      Coil( "Man_Tank_SirDolumVan_Ac" )
   END_RUNG
   // the same network as SCL:
   "Man_Tank_SirDolumVan_Ac" := "IN_Acil_stop" AND NOT "System".Auto_Man AND "HMI_Data".Buttons.ManuelButonlar.TankSirDolumVanasi_Ac;
END_REGION

REGION Network 2: Sirkiülasyon ve kalip vanasi kapat
   RUNG wire#powerrail
      Contact( "IN_Acil_stop" )
      Contact( "System".Auto_Man )
      Contact( "HMI_Data".Buttons.ManuelButonlar.SirKalipVanasi_Kapat )
      Coil( "Man_SirKalip_Van_Kapat" )
   END_RUNG
   // the same network as SCL:
   "Man_SirKalip_Van_Kapat" := "IN_Acil_stop" AND "System".Auto_Man AND "HMI_Data".Buttons.ManuelButonlar.SirKalipVanasi_Kapat;
END_REGION

REGION Network 3: Sirkiülasyon ve kalip vanasi ac
   RUNG wire#powerrail
      Contact( "IN_Acil_stop" )
      Contact( "System".Auto_Man )
      Contact( "HMI_Data".Buttons.ManuelButonlar.SirKalipVanasi_Ac )
      Coil( "Man_SirKalip_Van_Ac" )
   END_RUNG
   // the same network as SCL:
   "Man_SirKalip_Van_Ac" := "IN_Acil_stop" AND "System".Auto_Man AND "HMI_Data".Buttons.ManuelButonlar.SirKalipVanasi_Ac;
END_REGION

REGION Network 4: Baypass vanasi 1 kapat
   RUNG wire#powerrail
      Contact( "IN_Acil_stop" )
      Contact( "System".Auto_Man )
      Contact( "HMI_Data".Buttons.ManuelButonlar.BaypassVanasi1_Kapat )
      Coil( "Man_Baypass_Van_Kapat" )
   END_RUNG
   // the same network as SCL:
   "Man_Baypass_Van_Kapat" := "IN_Acil_stop" AND "System".Auto_Man AND "HMI_Data".Buttons.ManuelButonlar.BaypassVanasi1_Kapat;
END_REGION

REGION Network 5: Baypass vanasi 1 ac
   RUNG wire#powerrail
      Contact( "IN_Acil_stop" )
      Contact( "System".Auto_Man )
      Contact( "HMI_Data".Buttons.ManuelButonlar.BaypassVanasi1_Ac )
      Coil( "Man_Baypass_Van_Ac" )
   END_RUNG
   // the same network as SCL:
   "Man_Baypass_Van_Ac" := "IN_Acil_stop" AND "System".Auto_Man AND "HMI_Data".Buttons.ManuelButonlar.BaypassVanasi1_Ac;
END_REGION

REGION Network 6: Baypas vanasi 2 kapat
   RUNG wire#powerrail
      Contact( "IN_Acil_stop" )
      Contact( "System".Auto_Man )
      Contact( "HMI_Data".Buttons.ManuelButonlar.BaypassVanasi2_Kapat )
      Coil( "Man_Baypass2_Van_Kapat" )
   END_RUNG
   // the same network as SCL:
   "Man_Baypass2_Van_Kapat" := "IN_Acil_stop" AND "System".Auto_Man AND "HMI_Data".Buttons.ManuelButonlar.BaypassVanasi2_Kapat;
END_REGION

REGION Network 7: Baypas vanasi 2 ac
   RUNG wire#powerrail
      Contact( "IN_Acil_stop" )
      Contact( "System".Auto_Man )
      Contact( "HMI_Data".Buttons.ManuelButonlar.BaypassVanasi2_Ac )
      Coil( "Man_Baypass2_Van_Ac" )
   END_RUNG
   // the same network as SCL:
   "Man_Baypass2_Van_Ac" := "IN_Acil_stop" AND "System".Auto_Man AND "HMI_Data".Buttons.ManuelButonlar.BaypassVanasi2_Ac;
END_REGION

REGION Network 8: Motor 1 run
   "Man_Motor1_Kontaktor" := "IN_Acil_stop" AND "System".Auto_Man AND "HMI_Data".Buttons.ManuelButonlar.Motor1_Run AND "IN_Termik";
   #Man_Motor1_Run_Timer(IN := "Man_Motor1_Kontaktor", PT := t#2s);   // TON
   "Man_Motor1_Run" := #Man_Motor1_Run_Timer.Q;
END_REGION

REGION Network 9: Motor 2 run
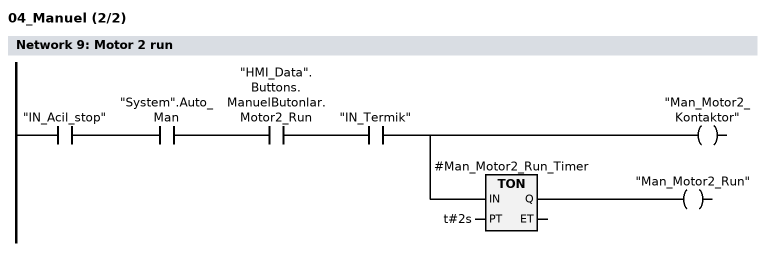
   "Man_Motor2_Kontaktor" := "IN_Acil_stop" AND "System".Auto_Man AND "HMI_Data".Buttons.ManuelButonlar.Motor2_Run AND "IN_Termik";
   #Man_Motor2_Run_Timer(IN := "Man_Motor2_Kontaktor", PT := t#2s);   // TON
   "Man_Motor2_Run" := #Man_Motor2_Run_Timer.Q;
END_REGION
END_FUNCTION_BLOCK

(* ===== HMI "HMI_RT_1" =====
system functions are stored by id; their names below are inferred from use
connection "HMI_Connection_1": ETHERNET, SMART_S7_1200_OMS

HMI tags "Default tag table"
   "HMI_Data_Infos.AnlikGirisSicakligi" : Real = PLC HMI_Data.Infos.AnlikGirisSicakligi, 1 s
   "HMI_Data_Infos.AnlikCikisSicakligi" : Real = PLC HMI_Data.Infos.AnlikCikisSicakligi, 1 s
   "HMI_Data_Datas.IstenenSicaklik" : Real = PLC HMI_Data.Datas.IstenenSicaklik, 1 s
   "HMI_Data_Infos.SystemDurumu" : String[50] = PLC HMI_Data.Infos.SystemDurumu, 1 s
   "HMI_Data_Buttons.Otomatik" : Bool = PLC HMI_Data.Buttons.Otomatik, 1 s
   "HMI_Data_Buttons.Manuel" : Bool = PLC HMI_Data.Buttons.Manuel, 1 s
   "HMI_Data_Buttons.Start" : Bool = PLC HMI_Data.Buttons.Start, 1 s
   "HMI_Data_Buttons.Stop" : Bool = PLC HMI_Data.Buttons.Stop, 1 s
   "HMI_Data_Buttons.AlarmSustur" : Bool = PLC HMI_Data.Buttons.AlarmSustur, 1 s
   "HMI_Data_Infos.FlowMeterOran" : Real = PLC HMI_Data.Infos.FlowMeterOran, 1 s
   "HMI_Data_Infos.OransalVanaOran" : Real = PLC HMI_Data.Infos.OransalVanaOran, 1 s
   "HMI_Data_Infos.yaslandirmaStatus.sol" : Bool = PLC HMI_Data.Infos.yaslandirmaStatus.sol, 1 s
   "HMI_Data_Infos.yaslandirmaStatus.sag" : Bool = PLC HMI_Data.Infos.yaslandirmaStatus.sag, 1 s
   "HMI_Data_Datas.driveSpeed" : Real = PLC HMI_Data.Datas.driveSpeed, 1 s
   "HMI_Data_Infos.driveActVelocity" : Real = PLC HMI_Data.Infos.driveActVelocity, 1 s
   "HMI_Data_Datas.istenenYaslandirmaSuresi_saat" : Int = PLC HMI_Data.Datas.istenenYaslandirmaSuresi_saat, 1 s
   "HMI_Data_Datas.istenenYaslandirmaSuresi_dk" : Int = PLC HMI_Data.Datas.istenenYaslandirmaSuresi_dk, 1 s
   "HMI_Data_Infos.yaslandirmaSuresi_saat" : DInt = PLC HMI_Data.Infos.yaslandirmaSuresi_saat, 1 s
   "HMI_Data_Infos.yaslandirmaSuresi_dk" : DInt = PLC HMI_Data.Infos.yaslandirmaSuresi_dk, 1 s
   "HMI_Data_Buttons.driveAckError" : Bool = PLC HMI_Data.Buttons.driveAckError, 1 s
   "IN_Termik" : Bool = PLC IN_Termik AT %I0.1, 1 s
   "HMI_Data_Datas.motorTercihi" : Byte = PLC HMI_Data.Datas.motorTercihi, 1 s
   "axisError" : Bool = PLC axisError AT %M30.2, 1 s

text list "Textlist_MotoSecimi": 0 'Her İkisi'; 1 'Motor 1'; 2 'Motor 2'

Template "Template_1" 480x272
   GraphicView "Logo" at 0,0 size 71x32; Picture "Logo of HMI_1"
   Button "Template_Button_1" at 2,231 size 91x34; TextOff 'Ana Menü'
      on Release: ActivateScreen("00_Root screen", 0)
   Button "Template_Button_2" at 98,231 size 91x34; TextOff 'Manuel'
      on Release: ActivateScreen("01_Manuel", 0)
   Button "Template_Button_3" at 195,231 size 91x34; TextOff 'Valf/Sensör'
      on Release: ActivateScreen("02_ValfBolumu", 0)
   Button "Template_Button_4" at 292,231 size 91x34; TextOff 'Yaşlandırma'
      on Release: ActivateScreen("03_Yaslandirma", 0)
   Button "Template_Button_5" at 386,231 size 91x34; TextOff 'Alarm'
      on Release: ActivateScreen("04_Alarm", 0)

Template "Template_2" 480x272
   Button "Template_Button_1" at 2,231 size 91x34; TextOff 'Ana Menü'
      on Release: ActivateScreen("00_Root screen", 0)
   Button "Template_Button_2" at 98,231 size 91x34; TextOff 'Manuel'
      on Release: ActivateScreen("01_Manuel", 0)
   Button "Template_Button_3" at 195,231 size 91x34; TextOff 'Valf/Sensör'
      on Release: ActivateScreen("02_ValfBolumu", 0)
   Button "Template_Button_4" at 292,231 size 91x34; TextOff 'Yaşlandırma'
      on Release: ActivateScreen("03_Yaslandirma", 0)
   Button "Template_Button_5" at 386,231 size 91x34; TextOff 'Alarm'
      on Release: ActivateScreen("04_Alarm", 0)

screen "00_Root screen" 480x272, template "Template_1"
   Button "Template_Button_1" at 57,68 size 149x39; TextOff 'Otomatik'
      on Press: function_b14e0dd5("HMI_Data_Buttons.Otomatik", 0)
   Button "Template_Button_2" at 269,67 size 149x39; TextOff 'Manuel'
      on Press: function_b14e0dd5("HMI_Data_Buttons.Manuel", 0)
   TextField "Text field_1" at 208,5 size 76x23; Text 'TCU-100'
   IOField "I/O field_1" at 1,35 size 478x28; FormatPattern ??????????????????????????????????????????????????
      ProcessValue <- "HMI_Data_Infos.SystemDurumu"
   Button "Template_Button_3" at 4,183 size 149x39; TextOff 'Start'
      on Press: function_b14e0dd5("HMI_Data_Buttons.Start", 0)
   Button "Template_Button_4" at 163,183 size 149x39; TextOff 'Stop'
      on Press: function_b14e0dd5("HMI_Data_Buttons.Stop", 0)
   IOField "I/O field_5" at 341,128 size 108x34; FormatPattern 999.9; Unit  C
      ProcessValue <- "HMI_Data_Datas.IstenenSicaklik"
   TextField "Text field_2" at 252,135 size 79x18; Text 'Sıcaklık Set:'
   IOField "I/O field_2" at 111,114 size 112x26; FormatPattern 9999.9; Unit  C
      ProcessValue <- "HMI_Data_Infos.AnlikGirisSicakligi"
   TextField "Text field_3" at 11,116 size 88x18; Text 'Giriş Sıcaklığı:'
   IOField "I/O field_3" at 111,148 size 112x26; FormatPattern 9999.9; Unit  C
      ProcessValue <- "HMI_Data_Infos.AnlikCikisSicakligi"
   TextField "Text field_4" at 11,150 size 89x18; Text 'Çıkış Sıcaklığı:'
   Button "Template_Button_5" at 324,183 size 149x39; TextOff 'Alarm Sustur'
      on Release: InvertBit("HMI_Data_Buttons.AlarmSustur")

screen "01_Manuel" 480x272, template "Template_2"
   Button "Button_1" at 363,182 size 110x43; TextOff 'Sayfa 2'
      on Release: ActivateScreen("01_Manuel2", 0)

screen "01_Manuel2" 480x272, template "Template_2"
   Button "Button_1" at 3,181 size 110x43; TextOff 'Geri'
      on Release: ActivateScreen("01_Manuel", 0)

screen "02_ValfBolumu" 480x272, template "Template_2"
   TextField "Text field_1" at 14,9 size 190x20; Text 'Sirkülasyon Tank Vanasi:'
   TextField "Text field_2" at 214,9 size 81x18; Text 'Sirkülasyon:'
   TextField "Text field_3" at 367,9 size 59x18; Text 'Su Alma:'
   TextField "Text field_4" at 32,47 size 138x38; Text 'Sirkülasyon/Kalıp Vanası'
   TextField "Text field_5" at 214,53 size 81x18; Text 'Sirkülasyon:'
   TextField "Text field_6" at 376,53 size 37x18; Text 'Kalıp:'
   Group "Group" at 1,89 size 477x44
   Group "Group_2" at 1,133 size 477x44
   Button "Button_1" at 363,182 size 110x43; TextOff 'Sayfa 2'
      on Release: ActivateScreen("02_ValfBolumu2", 0)
   TextField "Text field_7" at 49,98 size 118x20; Text 'Baypass Vanası'
   TextField "Text field_8" at 238,99 size 34x18; Text 'Açık:'
   TextField "Text field_9" at 372,99 size 45x18; Text 'Kapalı:'
   TextField "Text field_13" at 36,142 size 139x20; Text 'Tank Sıvı Seviyesi'
   TextField "Text field_14" at 238,141 size 33x18; Text 'Max:'
   TextField "Text field_15" at 379,141 size 30x18; Text 'Min:'

screen "02_ValfBolumu2" 480x272, template "Template_2"
   Button "Button_1" at 3,181 size 110x43; TextOff 'Geri'
      on Release: ActivateScreen("02_ValfBolumu", 0)
   TextField "Text field_1" at 91,9 size 117x20; Text 'Sıvı Akış Ölçer:'
   TextField "Text field_2" at 14,54 size 194x20; Text 'Oransal Vana Çıkış Oranı:'
   IOField "I/O field_2" at 216,8 size 169x27; FormatPattern 9999.99; Unit  %
      ProcessValue <- "HMI_Data_Infos.FlowMeterOran"
   IOField "I/O field_1" at 215,52 size 169x27; FormatPattern 9999.99; Unit  %
      ProcessValue <- "HMI_Data_Infos.OransalVanaOran"

screen "03_Yaslandirma" 480x272, template "Template_2"
   TextField "Text field_1" at 46,2 size 155x23; Text 'Yaşlandırma (Sol)'
   IOField "I/O field_5" at 169,75 size 125x27; FormatPattern 9999.9; Unit  %
      ProcessValue <- "HMI_Data_Datas.driveSpeed"
   TextField "Text field_6" at 20,79 size 141x18; Text 'Motor Hız Set Degeri:'
   IOField "I/O field_6" at 169,152 size 53x27; FormatPattern 99; Unit  s
      ProcessValue <- "HMI_Data_Datas.istenenYaslandirmaSuresi_saat"
   TextField "Text field_8" at 6,156 size 156x18; Text 'Yaşlandırma Set Süresi:'
   Circle "Circle_2" at 370,28 size 31x31
      Appearance <- "HMI_Data_Infos.yaslandirmaStatus.sag"
   TextField "Text field_9" at 317,34 size 38x18; Text 'Aktif:'
   TextField "Text field_10" at 278,2 size 160x23; Text 'Yaşlandırma (Sağ)'
   TextField "Text field_2" at 324,140 size 84x18; Text 'Termik Hata:'
   Circle "Circle_1" at 424,135 size 31x31
      Appearance <- "IN_Termik"
   TextField "Text field_3" at 6,197 size 155x18; Text 'Yaşlandırma Anlık Süre:'
   IOField "I/O field_1" at 169,194 size 53x27; FormatPattern 99; Unit  dk
      ProcessValue <- "HMI_Data_Infos.yaslandirmaSuresi_saat"
   TextField "Text field_4" at 340,74 size 92x18; Text 'Motor Tercihi:'
   SymbolicIOField "Symbolic I/O field_1" at 320,98 size 132x27; TextOn '1'; TextOff '0'; TextList "Textlist_MotoSecimi"
      ProcessValue <- "HMI_Data_Datas.motorTercihi"
   Button "Button_1" at 309,175 size 163x41; TextOff 'Motor Hata Reset'
      on Press: function_b14e0dd5("HMI_Data_Buttons.driveAckError", 0)
      Appearance <- "axisError"
   IOField "I/O field_2" at 169,113 size 124x27; FormatPattern 9999.9; Unit  %
      ProcessValue <- "HMI_Data_Infos.driveActVelocity"
   TextField "Text field_5" at 55,116 size 107x18; Text 'Anlık Motor Hızı:'
   Circle "Circle_3" at 137,28 size 31x31
      Appearance <- "HMI_Data_Infos.yaslandirmaStatus.sol"
   TextField "Text field_11" at 89,35 size 38x18; Text 'Aktif:'
   IOField "I/O field_3" at 228,152 size 65x27; FormatPattern 99; Unit  dk
      ProcessValue <- "HMI_Data_Datas.istenenYaslandirmaSuresi_dk"
   IOField "I/O field_4" at 228,194 size 64x27; FormatPattern 99; Unit  dk
      ProcessValue <- "HMI_Data_Infos.yaslandirmaSuresi_dk"

screen "04_Alarm" 480x272, template "Template_2"
   AlarmView "Alarm view_1" at 0,0 size 479x227
*)